KUKA KRL program: f1_Kuka_APT208T03S08.SRC

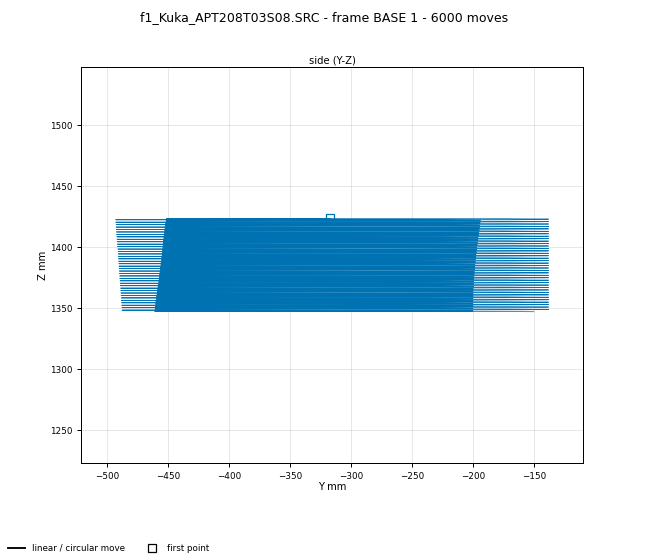
[picture p0: tool path of f1_Kuka_APT208T03S08.SRC in frame BASE 1, 6000 of 6001 moves have a stored position in this frame; points joined in program order, loops and branches not executed]
&ACCESS RVP
&REL 2
&PARAM TEMPLATE = C:\KRC\Roboter\Template\vorgabe
&PARAM EDITMASK = *
DEF f1_Kuka_APT208T03S08()


;FOLD INI;%{PE}%V3.2.0,%MKUKATPBASIS,%CINIT,%VCOMMON,%P
  ;FOLD BAS INI;%{E}%V3.2.0,%MKUKATPBASIS,%CINIT,%VINIT,%P
    GLOBAL INTERRUPT DECL 3 WHEN $STOPMESS==TRUE DO IR_STOPM ( )
    INTERRUPT ON 3
    BAS (#INITMOV,0 )
  ;ENDFOLD (BAS INI)
  ;FOLD USER INI;%{E}%V3.2.0,%MKUKATPUSER,%CINIT,%VINIT,%P
    ;Make your modifications here
  ;ENDFOLD (USER INI)
;ENDFOLD (INI)


;*** Make Null PTP Move
  PTP $pos_act

;*** Auto Load The Correct TOOL Data
  $tool=tool_data[3]

;*** Auto Load The Correct BASE Data
  $base=base_data[1]

  $ADVANCE = 5

;*** Restate Last Velocity
MMPM(30000.0)
SetRPM(6000)
LIN {X 0.078,Y -317.280,Z 1423.657,A 0.000,B 0.000,C 90.000,E1 298.281} C_DIS
LIN {X 0.027,Y -327.861,Z 1423.650,A 0.000,B 0.000,C 90.000,E1 297.052} C_DIS
LIN {X 0.042,Y -349.398,Z 1423.638,A 0.000,B 0.000,C 90.000,E1 294.771} C_DIS
LIN {X 0.137,Y -360.246,Z 1423.631,A 0.000,B 0.000,C 90.000,E1 293.643} C_DIS
LIN {X -0.205,Y -370.701,Z 1423.625,A 0.000,B 0.000,C 90.000,E1 292.589} C_DIS
LIN {X -0.139,Y -380.922,Z 1423.619,A 0.000,B 0.000,C 90.000,E1 291.461} C_DIS
LIN {X 0.117,Y -393.713,Z 1423.611,A 0.000,B 0.000,C 90.000,E1 289.993} C_DIS
LIN {X 0.075,Y -408.828,Z 1423.602,A 0.000,B 0.000,C 90.000,E1 288.308} C_DIS
LIN {X 0.018,Y -418.717,Z 1423.596,A 0.000,B 0.000,C 90.000,E1 287.221} C_DIS
LIN {X 0.155,Y -425.616,Z 1423.591,A 0.000,B 0.000,C 90.000,E1 286.386} C_DIS
LIN {X -0.080,Y -431.756,Z 1423.587,A 0.000,B 0.000,C 90.000,E1 285.607} C_DIS
LIN {X 0.159,Y -436.943,Z 1423.582,A 0.000,B 0.000,C 90.000,E1 284.773} C_DIS
LIN {X -0.092,Y -441.232,Z 1423.578,A 0.000,B 0.000,C 90.000,E1 284.008} C_DIS
LIN {X 0.232,Y -444.816,Z 1423.573,A 0.000,B 0.000,C 90.000,E1 283.175} C_DIS
LIN {X 0.051,Y -447.674,Z 1423.569,A 0.000,B 0.000,C 90.000,E1 282.411} C_DIS
LIN {X 0.083,Y -449.182,Z 1423.566,A 0.000,B 0.000,C 90.000,E1 281.883} C_DIS
LIN {X 0.037,Y -450.321,Z 1423.563,A 0.000,B 0.000,C 90.000,E1 281.366} C_DIS
LIN {X 0.091,Y -451.038,Z 1423.560,A 0.000,B 0.000,C 90.000,E1 280.838} C_DIS
LIN {X 0.150,Y -451.344,Z 1423.557,A 0.000,B 0.000,C 90.000,E1 280.310} C_DIS
LIN {X 0.133,Y -451.155,Z 1423.554,A 0.000,B 0.000,C 90.000,E1 279.792} C_DIS
LIN {X 0.195,Y -450.506,Z 1423.552,A 0.000,B 0.000,C 90.000,E1 279.265} C_DIS
LIN {X 0.182,Y -449.231,Z 1423.549,A 0.000,B 0.000,C 90.000,E1 278.746} C_DIS
LIN {X 0.234,Y -447.401,Z 1423.546,A 0.000,B 0.000,C 90.000,E1 278.219} C_DIS
LIN {X 0.210,Y -444.863,Z 1423.543,A 0.000,B 0.000,C 90.000,E1 277.701} C_DIS
LIN {X 0.172,Y -441.534,Z 1423.540,A 0.000,B 0.000,C 90.000,E1 277.182} C_DIS
LIN {X -0.047,Y -439.509,Z 1423.539,A 0.000,B 0.000,C 90.000,E1 276.947} C_DIS
LIN {X -0.110,Y -434.621,Z 1423.536,A 0.000,B 0.000,C 90.000,E1 276.429} C_DIS
LIN {X 0.045,Y -431.742,Z 1423.534,A 0.000,B 0.000,C 90.000,E1 276.144} C_DIS
LIN {X -0.110,Y -425.505,Z 1423.531,A 0.000,B 0.000,C 90.000,E1 275.682} C_DIS
LIN {X -0.196,Y -419.121,Z 1423.529,A 0.000,B 0.000,C 90.000,E1 275.277} C_DIS
LIN {X 0.069,Y -412.601,Z 1423.527,A 0.000,B 0.000,C 90.000,E1 274.878} C_DIS
LIN {X 0.054,Y -402.831,Z 1423.525,A 0.000,B 0.000,C 90.000,E1 274.416} C_DIS
LIN {X -0.018,Y -389.852,Z 1423.522,A 0.000,B 0.000,C 90.000,E1 273.898} C_DIS
LIN {X -0.100,Y -377.007,Z 1423.519,A 0.000,B 0.000,C 90.000,E1 273.440} C_DIS
LIN {X 0.045,Y -367.072,Z 1423.517,A 0.000,B 0.000,C 90.000,E1 273.094} C_DIS
LIN {X 0.073,Y -356.749,Z 1423.516,A 0.000,B 0.000,C 90.000,E1 272.808} C_DIS
LIN {X 0.056,Y -346.151,Z 1423.514,A 0.000,B 0.000,C 90.000,E1 272.579} C_DIS
LIN {X -0.061,Y -333.748,Z 1423.513,A 0.000,B 0.000,C 90.000,E1 272.407} C_DIS
LIN {X -0.117,Y -320.521,Z 1423.513,A 0.000,B 0.000,C 90.000,E1 272.293} C_DIS
LIN {X -0.070,Y -307.150,Z 1423.512,A 0.000,B 0.000,C 90.000,E1 272.236} C_DIS
LIN {X -0.069,Y -181.228,Z 1423.512,A 0.000,B 0.000,C 90.000,E1 272.236} C_DIS
LIN {X -0.066,Y -181.566,Z 1423.503,A 0.000,B 0.000,C 90.000,E1 270.516} C_DIS
LIN {X -0.076,Y -181.120,Z 1423.489,A 0.000,B 0.000,C 90.000,E1 267.993} C_DIS
LIN {X -0.088,Y -180.906,Z 1423.475,A 0.000,B 0.000,C 90.000,E1 265.469} C_DIS
LIN {X -0.031,Y -180.723,Z 1423.470,A 0.000,B 0.000,C 90.000,E1 264.609} C_DIS
LIN {X 0.066,Y -178.812,Z 1423.442,A 0.000,B 0.000,C 90.000,E1 259.511} C_DIS
LIN {X -0.026,Y -175.857,Z 1423.414,A 0.000,B 0.000,C 90.000,E1 254.448} C_DIS
LIN {X -0.045,Y -173.185,Z 1423.395,A 0.000,B 0.000,C 90.000,E1 251.040} C_DIS
LIN {X -0.042,Y -171.487,Z 1423.380,A 0.000,B 0.000,C 90.000,E1 248.465} C_DIS
LIN {X -0.054,Y -167.717,Z 1423.356,A 0.000,B 0.000,C 90.000,E1 244.152} C_DIS
LIN {X -0.038,Y -166.407,Z 1423.347,A 0.000,B 0.000,C 90.000,E1 242.410} C_DIS
LIN {X -0.040,Y -163.131,Z 1423.327,A 0.000,B 0.000,C 90.000,E1 238.918} C_DIS
LIN {X -0.074,Y -161.084,Z 1423.313,A 0.000,B 0.000,C 90.000,E1 236.294} C_DIS
LIN {X 0.036,Y -157.814,Z 1423.293,A 0.000,B 0.000,C 90.000,E1 232.718} C_DIS
LIN {X -0.026,Y -155.848,Z 1423.278,A 0.000,B 0.000,C 90.000,E1 230.070} C_DIS
LIN {X 0.031,Y -152.099,Z 1423.253,A 0.000,B 0.000,C 90.000,E1 225.567} C_DIS
LIN {X 0.049,Y -150.349,Z 1423.238,A 0.000,B 0.000,C 90.000,E1 222.852} C_DIS
LIN {X -0.022,Y -147.086,Z 1423.213,A 0.000,B 0.000,C 90.000,E1 218.338} C_DIS
LIN {X -0.027,Y -145.658,Z 1423.198,A 0.000,B 0.000,C 90.000,E1 215.598} C_DIS
LIN {X -0.024,Y -143.040,Z 1423.172,A 0.000,B 0.000,C 90.000,E1 211.003} C_DIS
LIN {X -0.023,Y -141.664,Z 1423.152,A 0.000,B 0.000,C 90.000,E1 207.308} C_DIS
LIN {X 0.022,Y -139.449,Z 1423.116,A 0.000,B 0.000,C 90.000,E1 200.791} C_DIS
LIN {X -0.058,Y -139.184,Z 1423.105,A 0.000,B 0.000,C 90.000,E1 198.960} C_DIS
LIN {X -0.034,Y -138.322,Z 1423.053,A 0.000,B 0.000,C 90.000,E1 189.613} C_DIS
LIN {X -0.027,Y -139.462,Z 1423.007,A 0.000,B 0.000,C 90.000,E1 181.203} C_DIS
LIN {X 0.053,Y -141.022,Z 1422.976,A 0.000,B 0.000,C 90.000,E1 175.584} C_DIS
LIN {X 0.007,Y -142.386,Z 1422.960,A 0.000,B 0.000,C 90.000,E1 172.818} C_DIS
LIN {X -0.072,Y -144.617,Z 1422.934,A 0.000,B 0.000,C 90.000,E1 168.229} C_DIS
LIN {X -0.010,Y -147.812,Z 1422.909,A 0.000,B 0.000,C 90.000,E1 163.614} C_DIS
LIN {X 0.077,Y -150.499,Z 1422.889,A 0.000,B 0.000,C 90.000,E1 159.934} C_DIS
LIN {X -0.043,Y -153.958,Z 1422.869,A 0.000,B 0.000,C 90.000,E1 156.357} C_DIS
LIN {X 0.019,Y -157.369,Z 1422.849,A 0.000,B 0.000,C 90.000,E1 152.743} C_DIS
LIN {X -0.038,Y -161.569,Z 1422.829,A 0.000,B 0.000,C 90.000,E1 149.203} C_DIS
LIN {X -0.027,Y -165.767,Z 1422.809,A 0.000,B 0.000,C 90.000,E1 145.674} C_DIS
LIN {X -0.040,Y -170.725,Z 1422.790,A 0.000,B 0.000,C 90.000,E1 142.190} C_DIS
LIN {X 0.002,Y -175.598,Z 1422.771,A 0.000,B 0.000,C 90.000,E1 138.728} C_DIS
LIN {X -0.011,Y -181.215,Z 1422.752,A 0.000,B 0.000,C 90.000,E1 135.324} C_DIS
LIN {X -0.019,Y -186.679,Z 1422.733,A 0.000,B 0.000,C 90.000,E1 131.962} C_DIS
LIN {X -0.075,Y -191.282,Z 1422.719,A 0.000,B 0.000,C 90.000,E1 129.483} C_DIS
LIN {X 0.005,Y -197.107,Z 1422.701,A 0.000,B 0.000,C 90.000,E1 126.171} C_DIS
LIN {X 0.026,Y -199.962,Z 1422.693,A 0.000,B 0.000,C 90.000,E1 124.739} C_DIS
LIN {X 0.006,Y -311.159,Z 1422.693,A 0.000,B 0.000,C 90.000,E1 124.739} C_DIS
LIN {X -0.064,Y -312.139,Z 1422.693,A 0.000,B 0.000,C 90.000,E1 124.739} C_DIS
LIN {X 0.065,Y -316.789,Z 1422.692,A 0.000,B 0.000,C 90.000,E1 124.532} C_DIS
LIN {X 0.109,Y -319.895,Z 1422.691,A 0.000,B 0.000,C 90.000,E1 124.278} C_DIS
LIN {X 0.005,Y -323.594,Z 1422.688,A 0.000,B 0.000,C 90.000,E1 123.833} C_DIS
LIN {X 0.086,Y -325.369,Z 1422.686,A 0.000,B 0.000,C 90.000,E1 123.499} C_DIS
LIN {X 0.169,Y -326.751,Z 1422.684,A 0.000,B 0.000,C 90.000,E1 123.166} C_DIS
LIN {X 0.039,Y -338.501,Z 1422.667,A 0.000,B 0.000,C 90.000,E1 120.050} C_DIS
LIN {X 0.192,Y -350.479,Z 1422.652,A 0.000,B 0.000,C 90.000,E1 117.257} C_DIS
LIN {X -0.102,Y -363.919,Z 1422.636,A 0.000,B 0.000,C 90.000,E1 114.591} C_DIS
LIN {X 0.056,Y -377.182,Z 1422.623,A 0.000,B 0.000,C 90.000,E1 112.206} C_DIS
LIN {X 0.128,Y -391.780,Z 1422.611,A 0.000,B 0.000,C 90.000,E1 109.885} C_DIS
LIN {X 0.065,Y -407.816,Z 1422.598,A 0.000,B 0.000,C 90.000,E1 107.638} C_DIS
LIN {X 0.145,Y -425.401,Z 1422.586,A 0.000,B 0.000,C 90.000,E1 105.426} C_DIS
LIN {X 0.053,Y -444.616,Z 1422.574,A 0.000,B 0.000,C 90.000,E1 103.300} C_DIS
LIN {X 0.107,Y -464.726,Z 1422.563,A 0.000,B 0.000,C 90.000,E1 101.299} C_DIS
LIN {X -0.177,Y -485.356,Z 1422.553,A 0.000,B 0.000,C 90.000,E1 99.500} C_DIS
LIN {X -0.056,Y -487.492,Z 1422.551,A 0.000,B 0.000,C 90.000,E1 99.265} C_DIS
LIN {X 0.065,Y -489.116,Z 1422.550,A 0.000,B 0.000,C 90.000,E1 99.029} C_DIS
LIN {X -0.113,Y -490.499,Z 1422.549,A 0.000,B 0.000,C 90.000,E1 98.803} C_DIS
LIN {X -0.215,Y -491.522,Z 1422.547,A 0.000,B 0.000,C 90.000,E1 98.568} C_DIS
LIN {X 0.009,Y -492.685,Z 1422.545,A 0.000,B 0.000,C 90.000,E1 98.049} C_DIS
LIN {X -0.247,Y -492.827,Z 1422.542,A 0.000,B 0.000,C 90.000,E1 97.587} C_DIS
LIN {X -0.007,Y -491.972,Z 1422.539,A 0.000,B 0.000,C 90.000,E1 97.068} C_DIS
LIN {X -0.253,Y -489.975,Z 1422.536,A 0.000,B 0.000,C 90.000,E1 96.606} C_DIS
LIN {X 0.196,Y -483.357,Z 1422.531,A 0.000,B 0.000,C 90.000,E1 95.568} C_DIS
LIN {X 0.126,Y -469.087,Z 1422.519,A 0.000,B 0.000,C 90.000,E1 93.326} C_DIS
LIN {X 0.072,Y -460.783,Z 1422.511,A 0.000,B 0.000,C 90.000,E1 92.064} C_DIS
LIN {X -0.021,Y -440.905,Z 1422.494,A 0.000,B 0.000,C 90.000,E1 88.969} C_DIS
LIN {X -0.162,Y -429.949,Z 1422.484,A 0.000,B 0.000,C 90.000,E1 87.135} C_DIS
LIN {X -0.076,Y -418.773,Z 1422.474,A 0.000,B 0.000,C 90.000,E1 85.241} C_DIS
LIN {X -0.085,Y -405.939,Z 1422.461,A 0.000,B 0.000,C 90.000,E1 83.053} C_DIS
LIN {X 0.034,Y -394.598,Z 1422.450,A 0.000,B 0.000,C 90.000,E1 81.084} C_DIS
LIN {X -0.016,Y -383.087,Z 1422.439,A 0.000,B 0.000,C 90.000,E1 79.106} C_DIS
LIN {X 0.130,Y -371.680,Z 1422.428,A 0.000,B 0.000,C 90.000,E1 77.061} C_DIS
LIN {X -0.149,Y -360.358,Z 1422.417,A 0.000,B 0.000,C 90.000,E1 75.046} C_DIS
LIN {X 0.121,Y -349.003,Z 1422.405,A 0.000,B 0.000,C 90.000,E1 72.906} C_DIS
LIN {X 0.016,Y -339.072,Z 1422.395,A 0.000,B 0.000,C 90.000,E1 71.094} C_DIS
LIN {X 0.102,Y -325.927,Z 1422.381,A 0.000,B 0.000,C 90.000,E1 68.592} C_DIS
LIN {X -0.007,Y -308.641,Z 1422.362,A 0.000,B 0.000,C 90.000,E1 65.101} C_DIS
LIN {X -0.028,Y -295.960,Z 1422.345,A 0.000,B 0.000,C 90.000,E1 62.153} C_DIS
LIN {X 0.004,Y -283.341,Z 1422.327,A 0.000,B 0.000,C 90.000,E1 58.791} C_DIS
LIN {X -0.145,Y -271.830,Z 1422.307,A 0.000,B 0.000,C 90.000,E1 55.388} C_DIS
LIN {X 0.077,Y -262.146,Z 1422.290,A 0.000,B 0.000,C 90.000,E1 52.190} C_DIS
LIN {X -0.025,Y -252.090,Z 1422.270,A 0.000,B 0.000,C 90.000,E1 48.647} C_DIS
LIN {X 0.025,Y -242.796,Z 1422.250,A 0.000,B 0.000,C 90.000,E1 45.000} C_DIS
LIN {X -0.027,Y -234.404,Z 1422.229,A 0.000,B 0.000,C 90.000,E1 41.310} C_DIS
LIN {X 0.060,Y -226.842,Z 1422.208,A 0.000,B 0.000,C 90.000,E1 37.523} C_DIS
LIN {X 0.036,Y -220.187,Z 1422.187,A 0.000,B 0.000,C 90.000,E1 33.706} C_DIS
LIN {X -0.122,Y -214.311,Z 1422.166,A 0.000,B 0.000,C 90.000,E1 29.873} C_DIS
LIN {X -0.025,Y -209.279,Z 1422.144,A 0.000,B 0.000,C 90.000,E1 25.924} C_DIS
LIN {X -0.066,Y -205.139,Z 1422.122,A 0.000,B 0.000,C 90.000,E1 21.972} C_DIS
LIN {X 0.010,Y -201.303,Z 1422.095,A 0.000,B 0.000,C 90.000,E1 17.149} C_DIS
LIN {X 0.047,Y -198.459,Z 1422.068,A 0.000,B 0.000,C 90.000,E1 12.299} C_DIS
LIN {X 0.088,Y -196.155,Z 1422.037,A 0.000,B 0.000,C 90.000,E1 6.606} C_DIS
LIN {X 0.027,Y -194.653,Z 1422.005,A 0.000,B 0.000,C 90.000,E1 0.917} C_DIS
LIN {X 0.004,Y -194.202,Z 1421.984,A 0.000,B 0.000,C 90.000,E1 357.078} C_DIS
LIN {X -0.051,Y -194.204,Z 1421.957,A 0.000,B 0.000,C 90.000,E1 352.186} C_DIS
LIN {X -0.046,Y -195.369,Z 1421.920,A 0.000,B 0.000,C 90.000,E1 345.644} C_DIS
LIN {X -0.018,Y -198.094,Z 1421.889,A 0.000,B 0.000,C 90.000,E1 339.934} C_DIS
LIN {X -0.100,Y -202.039,Z 1421.862,A 0.000,B 0.000,C 90.000,E1 335.101} C_DIS
LIN {X 0.034,Y -206.546,Z 1421.839,A 0.000,B 0.000,C 90.000,E1 331.051} C_DIS
LIN {X 0.048,Y -210.949,Z 1421.822,A 0.000,B 0.000,C 90.000,E1 327.867} C_DIS
LIN {X -0.018,Y -216.341,Z 1421.804,A 0.000,B 0.000,C 90.000,E1 324.736} C_DIS
LIN {X 0.002,Y -222.667,Z 1421.787,A 0.000,B 0.000,C 90.000,E1 321.618} C_DIS
LIN {X -0.075,Y -229.928,Z 1421.770,A 0.000,B 0.000,C 90.000,E1 318.566} C_DIS
LIN {X -0.029,Y -239.211,Z 1421.751,A 0.000,B 0.000,C 90.000,E1 315.162} C_DIS
LIN {X -0.040,Y -249.686,Z 1421.732,A 0.000,B 0.000,C 90.000,E1 311.838} C_DIS
LIN {X 0.098,Y -260.059,Z 1421.716,A 0.000,B 0.000,C 90.000,E1 308.910} C_DIS
LIN {X 0.021,Y -271.627,Z 1421.701,A 0.000,B 0.000,C 90.000,E1 306.091} C_DIS
LIN {X 0.083,Y -281.387,Z 1421.689,A 0.000,B 0.000,C 90.000,E1 303.992} C_DIS
LIN {X 0.073,Y -288.584,Z 1421.681,A 0.000,B 0.000,C 90.000,E1 302.625} C_DIS
LIN {X 0.154,Y -296.526,Z 1421.674,A 0.000,B 0.000,C 90.000,E1 301.258} C_DIS
LIN {X 0.029,Y -305.181,Z 1421.666,A 0.000,B 0.000,C 90.000,E1 299.951} C_DIS
LIN {X 0.166,Y -314.744,Z 1421.659,A 0.000,B 0.000,C 90.000,E1 298.615} C_DIS
LIN {X 0.045,Y -325.085,Z 1421.652,A 0.000,B 0.000,C 90.000,E1 297.385} C_DIS
LIN {X 0.084,Y -346.523,Z 1421.639,A 0.000,B 0.000,C 90.000,E1 295.079} C_DIS
LIN {X 0.154,Y -359.883,Z 1421.632,A 0.000,B 0.000,C 90.000,E1 293.695} C_DIS
LIN {X -0.165,Y -370.313,Z 1421.626,A 0.000,B 0.000,C 90.000,E1 292.642} C_DIS
LIN {X 0.087,Y -380.561,Z 1421.619,A 0.000,B 0.000,C 90.000,E1 291.482} C_DIS
LIN {X 0.001,Y -393.292,Z 1421.611,A 0.000,B 0.000,C 90.000,E1 290.066} C_DIS
LIN {X 0.132,Y -408.362,Z 1421.602,A 0.000,B 0.000,C 90.000,E1 288.362} C_DIS
LIN {X -0.004,Y -418.330,Z 1421.596,A 0.000,B 0.000,C 90.000,E1 287.275} C_DIS
LIN {X -0.191,Y -425.234,Z 1421.592,A 0.000,B 0.000,C 90.000,E1 286.496} C_DIS
LIN {X -0.022,Y -431.464,Z 1421.587,A 0.000,B 0.000,C 90.000,E1 285.662} C_DIS
LIN {X -0.089,Y -435.100,Z 1421.584,A 0.000,B 0.000,C 90.000,E1 285.134} C_DIS
LIN {X 0.182,Y -439.765,Z 1421.580,A 0.000,B 0.000,C 90.000,E1 284.300} C_DIS
LIN {X -0.044,Y -443.624,Z 1421.575,A 0.000,B 0.000,C 90.000,E1 283.536} C_DIS
LIN {X -0.029,Y -445.806,Z 1421.572,A 0.000,B 0.000,C 90.000,E1 283.008} C_DIS
LIN {X 0.001,Y -447.703,Z 1421.569,A 0.000,B 0.000,C 90.000,E1 282.479} C_DIS
LIN {X 0.037,Y -449.267,Z 1421.566,A 0.000,B 0.000,C 90.000,E1 281.951} C_DIS
LIN {X 0.082,Y -450.452,Z 1421.563,A 0.000,B 0.000,C 90.000,E1 281.422} C_DIS
LIN {X 0.137,Y -451.260,Z 1421.561,A 0.000,B 0.000,C 90.000,E1 280.894} C_DIS
LIN {X 0.196,Y -451.636,Z 1421.558,A 0.000,B 0.000,C 90.000,E1 280.366} C_DIS
LIN {X 0.179,Y -451.549,Z 1421.555,A 0.000,B 0.000,C 90.000,E1 279.849} C_DIS
LIN {X 0.242,Y -450.932,Z 1421.552,A 0.000,B 0.000,C 90.000,E1 279.321} C_DIS
LIN {X -0.214,Y -449.794,Z 1421.549,A 0.000,B 0.000,C 90.000,E1 278.859} C_DIS
LIN {X -0.224,Y -448.053,Z 1421.546,A 0.000,B 0.000,C 90.000,E1 278.341} C_DIS
LIN {X -0.178,Y -445.618,Z 1421.543,A 0.000,B 0.000,C 90.000,E1 277.814} C_DIS
LIN {X -0.210,Y -442.391,Z 1421.540,A 0.000,B 0.000,C 90.000,E1 277.296} C_DIS
LIN {X 0.011,Y -440.500,Z 1421.539,A 0.000,B 0.000,C 90.000,E1 277.004} C_DIS
LIN {X -0.049,Y -435.790,Z 1421.536,A 0.000,B 0.000,C 90.000,E1 276.486} C_DIS
LIN {X 0.109,Y -433.033,Z 1421.535,A 0.000,B 0.000,C 90.000,E1 276.201} C_DIS
LIN {X -0.144,Y -426.825,Z 1421.532,A 0.000,B 0.000,C 90.000,E1 275.739} C_DIS
LIN {X 0.107,Y -420.413,Z 1421.529,A 0.000,B 0.000,C 90.000,E1 275.277} C_DIS
LIN {X -0.107,Y -413.942,Z 1421.527,A 0.000,B 0.000,C 90.000,E1 274.935} C_DIS
LIN {X 0.054,Y -407.470,Z 1421.526,A 0.000,B 0.000,C 90.000,E1 274.588} C_DIS
LIN {X -0.116,Y -397.720,Z 1421.523,A 0.000,B 0.000,C 90.000,E1 274.188} C_DIS
LIN {X 0.001,Y -384.828,Z 1421.520,A 0.000,B 0.000,C 90.000,E1 273.669} C_DIS
LIN {X 0.050,Y -371.840,Z 1421.518,A 0.000,B 0.000,C 90.000,E1 273.212} C_DIS
LIN {X -0.033,Y -361.640,Z 1421.516,A 0.000,B 0.000,C 90.000,E1 272.922} C_DIS
LIN {X -0.159,Y -350.920,Z 1421.515,A 0.000,B 0.000,C 90.000,E1 272.694} C_DIS
LIN {X 0.014,Y -343.452,Z 1421.514,A 0.000,B 0.000,C 90.000,E1 272.522} C_DIS
LIN {X -0.054,Y -335.045,Z 1421.513,A 0.000,B 0.000,C 90.000,E1 272.407} C_DIS
LIN {X -0.110,Y -321.941,Z 1421.513,A 0.000,B 0.000,C 90.000,E1 272.293} C_DIS
LIN {X -0.069,Y -310.020,Z 1421.512,A 0.000,B 0.000,C 90.000,E1 272.236} C_DIS
LIN {X -0.069,Y -181.228,Z 1421.512,A 0.000,B 0.000,C 90.000,E1 272.236} C_DIS
LIN {X -0.072,Y -181.566,Z 1421.503,A 0.000,B 0.000,C 90.000,E1 270.516} C_DIS
LIN {X -0.082,Y -181.119,Z 1421.489,A 0.000,B 0.000,C 90.000,E1 267.993} C_DIS
LIN {X 0.087,Y -180.907,Z 1421.475,A 0.000,B 0.000,C 90.000,E1 265.412} C_DIS
LIN {X -0.036,Y -180.723,Z 1421.470,A 0.000,B 0.000,C 90.000,E1 264.609} C_DIS
LIN {X 0.061,Y -178.811,Z 1421.442,A 0.000,B 0.000,C 90.000,E1 259.511} C_DIS
LIN {X -0.032,Y -175.856,Z 1421.414,A 0.000,B 0.000,C 90.000,E1 254.448} C_DIS
LIN {X -0.050,Y -173.184,Z 1421.395,A 0.000,B 0.000,C 90.000,E1 251.040} C_DIS
LIN {X -0.048,Y -171.486,Z 1421.380,A 0.000,B 0.000,C 90.000,E1 248.465} C_DIS
LIN {X -0.060,Y -167.715,Z 1421.356,A 0.000,B 0.000,C 90.000,E1 244.152} C_DIS
LIN {X -0.044,Y -166.406,Z 1421.347,A 0.000,B 0.000,C 90.000,E1 242.410} C_DIS
LIN {X -0.045,Y -163.130,Z 1421.327,A 0.000,B 0.000,C 90.000,E1 238.918} C_DIS
LIN {X -0.079,Y -161.082,Z 1421.313,A 0.000,B 0.000,C 90.000,E1 236.294} C_DIS
LIN {X 0.031,Y -157.812,Z 1421.293,A 0.000,B 0.000,C 90.000,E1 232.718} C_DIS
LIN {X -0.031,Y -155.847,Z 1421.278,A 0.000,B 0.000,C 90.000,E1 230.070} C_DIS
LIN {X 0.025,Y -152.097,Z 1421.253,A 0.000,B 0.000,C 90.000,E1 225.567} C_DIS
LIN {X 0.044,Y -150.348,Z 1421.238,A 0.000,B 0.000,C 90.000,E1 222.852} C_DIS
LIN {X -0.027,Y -147.085,Z 1421.213,A 0.000,B 0.000,C 90.000,E1 218.338} C_DIS
LIN {X -0.032,Y -145.657,Z 1421.198,A 0.000,B 0.000,C 90.000,E1 215.598} C_DIS
LIN {X -0.029,Y -143.040,Z 1421.172,A 0.000,B 0.000,C 90.000,E1 211.003} C_DIS
LIN {X -0.028,Y -141.664,Z 1421.152,A 0.000,B 0.000,C 90.000,E1 207.308} C_DIS
LIN {X 0.017,Y -139.449,Z 1421.116,A 0.000,B 0.000,C 90.000,E1 200.791} C_DIS
LIN {X 0.069,Y -139.183,Z 1421.105,A 0.000,B 0.000,C 90.000,E1 198.906} C_DIS
LIN {X -0.039,Y -138.321,Z 1421.053,A 0.000,B 0.000,C 90.000,E1 189.613} C_DIS
LIN {X -0.032,Y -139.463,Z 1421.007,A 0.000,B 0.000,C 90.000,E1 181.203} C_DIS
LIN {X 0.048,Y -141.023,Z 1420.976,A 0.000,B 0.000,C 90.000,E1 175.584} C_DIS
LIN {X 0.003,Y -142.387,Z 1420.960,A 0.000,B 0.000,C 90.000,E1 172.818} C_DIS
LIN {X 0.065,Y -144.619,Z 1420.934,A 0.000,B 0.000,C 90.000,E1 168.173} C_DIS
LIN {X -0.015,Y -147.812,Z 1420.909,A 0.000,B 0.000,C 90.000,E1 163.614} C_DIS
LIN {X 0.073,Y -150.501,Z 1420.889,A 0.000,B 0.000,C 90.000,E1 159.934} C_DIS
LIN {X -0.048,Y -153.960,Z 1420.869,A 0.000,B 0.000,C 90.000,E1 156.357} C_DIS
LIN {X 0.015,Y -157.371,Z 1420.849,A 0.000,B 0.000,C 90.000,E1 152.743} C_DIS
LIN {X -0.044,Y -161.572,Z 1420.829,A 0.000,B 0.000,C 90.000,E1 149.203} C_DIS
LIN {X -0.032,Y -165.769,Z 1420.809,A 0.000,B 0.000,C 90.000,E1 145.674} C_DIS
LIN {X -0.045,Y -170.728,Z 1420.790,A 0.000,B 0.000,C 90.000,E1 142.190} C_DIS
LIN {X -0.002,Y -175.600,Z 1420.771,A 0.000,B 0.000,C 90.000,E1 138.728} C_DIS
LIN {X -0.016,Y -181.217,Z 1420.752,A 0.000,B 0.000,C 90.000,E1 135.324} C_DIS
LIN {X -0.024,Y -186.683,Z 1420.733,A 0.000,B 0.000,C 90.000,E1 131.962} C_DIS
LIN {X -0.081,Y -191.285,Z 1420.719,A 0.000,B 0.000,C 90.000,E1 129.483} C_DIS
LIN {X -0.001,Y -197.110,Z 1420.701,A 0.000,B 0.000,C 90.000,E1 126.171} C_DIS
LIN {X -0.021,Y -199.922,Z 1420.693,A 0.000,B 0.000,C 90.000,E1 124.771} C_DIS
LIN {X 0.108,Y -311.246,Z 1420.693,A 0.000,B 0.000,C 90.000,E1 124.739} C_DIS
LIN {X 0.056,Y -317.044,Z 1420.692,A 0.000,B 0.000,C 90.000,E1 124.532} C_DIS
LIN {X 0.084,Y -320.054,Z 1420.691,A 0.000,B 0.000,C 90.000,E1 124.278} C_DIS
LIN {X 0.154,Y -323.760,Z 1420.688,A 0.000,B 0.000,C 90.000,E1 123.785} C_DIS
LIN {X -0.033,Y -325.477,Z 1420.686,A 0.000,B 0.000,C 90.000,E1 123.499} C_DIS
LIN {X -0.125,Y -327.926,Z 1420.682,A 0.000,B 0.000,C 90.000,E1 122.880} C_DIS
LIN {X -0.082,Y -338.563,Z 1420.667,A 0.000,B 0.000,C 90.000,E1 120.050} C_DIS
LIN {X 0.067,Y -350.550,Z 1420.651,A 0.000,B 0.000,C 90.000,E1 117.257} C_DIS
LIN {X -0.077,Y -364.001,Z 1420.636,A 0.000,B 0.000,C 90.000,E1 114.567} C_DIS
LIN {X -0.073,Y -377.275,Z 1420.623,A 0.000,B 0.000,C 90.000,E1 112.206} C_DIS
LIN {X -0.003,Y -391.885,Z 1420.610,A 0.000,B 0.000,C 90.000,E1 109.885} C_DIS
LIN {X -0.070,Y -407.932,Z 1420.598,A 0.000,B 0.000,C 90.000,E1 107.638} C_DIS
LIN {X 0.007,Y -425.531,Z 1420.586,A 0.000,B 0.000,C 90.000,E1 105.426} C_DIS
LIN {X -0.086,Y -444.758,Z 1420.574,A 0.000,B 0.000,C 90.000,E1 103.300} C_DIS
LIN {X -0.027,Y -464.873,Z 1420.563,A 0.000,B 0.000,C 90.000,E1 101.299} C_DIS
LIN {X 0.172,Y -485.485,Z 1420.553,A 0.000,B 0.000,C 90.000,E1 99.443} C_DIS
LIN {X -0.196,Y -487.560,Z 1420.551,A 0.000,B 0.000,C 90.000,E1 99.265} C_DIS
LIN {X -0.085,Y -489.142,Z 1420.550,A 0.000,B 0.000,C 90.000,E1 99.029} C_DIS
LIN {X -0.263,Y -490.481,Z 1420.549,A 0.000,B 0.000,C 90.000,E1 98.803} C_DIS
LIN {X 0.120,Y -491.469,Z 1420.547,A 0.000,B 0.000,C 90.000,E1 98.511} C_DIS
LIN {X -0.142,Y -492.573,Z 1420.545,A 0.000,B 0.000,C 90.000,E1 98.049} C_DIS
LIN {X 0.091,Y -492.661,Z 1420.542,A 0.000,B 0.000,C 90.000,E1 97.530} C_DIS
LIN {X -0.158,Y -491.750,Z 1420.539,A 0.000,B 0.000,C 90.000,E1 97.068} C_DIS
LIN {X 0.082,Y -489.682,Z 1420.536,A 0.000,B 0.000,C 90.000,E1 96.549} C_DIS
LIN {X -0.119,Y -471.909,Z 1420.521,A 0.000,B 0.000,C 90.000,E1 93.841} C_DIS
LIN {X 0.066,Y -465.501,Z 1420.516,A 0.000,B 0.000,C 90.000,E1 92.808} C_DIS
LIN {X -0.035,Y -453.683,Z 1420.506,A 0.000,B 0.000,C 90.000,E1 91.031} C_DIS
LIN {X -0.087,Y -435.958,Z 1420.490,A 0.000,B 0.000,C 90.000,E1 88.165} C_DIS
LIN {X -0.159,Y -428.109,Z 1420.482,A 0.000,B 0.000,C 90.000,E1 86.846} C_DIS
LIN {X 0.177,Y -418.551,Z 1420.473,A 0.000,B 0.000,C 90.000,E1 85.184} C_DIS
LIN {X 0.153,Y -405.740,Z 1420.461,A 0.000,B 0.000,C 90.000,E1 82.996} C_DIS
LIN {X -0.203,Y -396.035,Z 1420.452,A 0.000,B 0.000,C 90.000,E1 81.376} C_DIS
LIN {X 0.112,Y -386.226,Z 1420.443,A 0.000,B 0.000,C 90.000,E1 79.634} C_DIS
LIN {X -0.034,Y -373.150,Z 1420.430,A 0.000,B 0.000,C 90.000,E1 77.353} C_DIS
LIN {X 0.069,Y -361.829,Z 1420.418,A 0.000,B 0.000,C 90.000,E1 75.283} C_DIS
LIN {X 0.036,Y -350.461,Z 1420.407,A 0.000,B 0.000,C 90.000,E1 73.196} C_DIS
LIN {X -0.144,Y -340.573,Z 1420.396,A 0.000,B 0.000,C 90.000,E1 71.402} C_DIS
LIN {X -0.018,Y -327.372,Z 1420.383,A 0.000,B 0.000,C 90.000,E1 68.901} C_DIS
LIN {X -0.077,Y -309.930,Z 1420.363,A 0.000,B 0.000,C 90.000,E1 65.409} C_DIS
LIN {X 0.075,Y -297.134,Z 1420.347,A 0.000,B 0.000,C 90.000,E1 62.436} C_DIS
LIN {X -0.098,Y -285.611,Z 1420.330,A 0.000,B 0.000,C 90.000,E1 59.459} C_DIS
LIN {X 0.056,Y -273.952,Z 1420.311,A 0.000,B 0.000,C 90.000,E1 56.008} C_DIS
LIN {X -0.034,Y -264.211,Z 1420.294,A 0.000,B 0.000,C 90.000,E1 52.889} C_DIS
LIN {X 0.137,Y -254.008,Z 1420.274,A 0.000,B 0.000,C 90.000,E1 49.299} C_DIS
LIN {X -0.090,Y -244.588,Z 1420.254,A 0.000,B 0.000,C 90.000,E1 45.729} C_DIS
LIN {X 0.077,Y -236.040,Z 1420.233,A 0.000,B 0.000,C 90.000,E1 42.000} C_DIS
LIN {X 0.036,Y -228.338,Z 1420.213,A 0.000,B 0.000,C 90.000,E1 38.257} C_DIS
LIN {X 0.009,Y -221.529,Z 1420.191,A 0.000,B 0.000,C 90.000,E1 34.452} C_DIS
LIN {X -0.002,Y -215.542,Z 1420.170,A 0.000,B 0.000,C 90.000,E1 30.590} C_DIS
LIN {X 0.036,Y -210.353,Z 1420.148,A 0.000,B 0.000,C 90.000,E1 26.668} C_DIS
LIN {X 0.019,Y -206.069,Z 1420.126,A 0.000,B 0.000,C 90.000,E1 22.717} C_DIS
LIN {X -0.055,Y -202.099,Z 1420.100,A 0.000,B 0.000,C 90.000,E1 17.946} C_DIS
LIN {X -0.070,Y -199.183,Z 1420.073,A 0.000,B 0.000,C 90.000,E1 13.119} C_DIS
LIN {X 0.069,Y -197.011,Z 1420.046,A 0.000,B 0.000,C 90.000,E1 8.219} C_DIS
LIN {X -0.018,Y -195.935,Z 1420.028,A 0.000,B 0.000,C 90.000,E1 4.992} C_DIS
LIN {X -0.035,Y -194.777,Z 1419.997,A 0.000,B 0.000,C 90.000,E1 359.542} C_DIS
LIN {X 0.067,Y -194.386,Z 1419.970,A 0.000,B 0.000,C 90.000,E1 354.609} C_DIS
LIN {X -0.054,Y -194.593,Z 1419.947,A 0.000,B 0.000,C 90.000,E1 350.557} C_DIS
LIN {X -0.011,Y -196.562,Z 1419.907,A 0.000,B 0.000,C 90.000,E1 343.196} C_DIS
LIN {X 0.079,Y -200.084,Z 1419.875,A 0.000,B 0.000,C 90.000,E1 337.486} C_DIS
LIN {X 0.064,Y -203.944,Z 1419.853,A 0.000,B 0.000,C 90.000,E1 333.461} C_DIS
LIN {X 0.091,Y -208.830,Z 1419.830,A 0.000,B 0.000,C 90.000,E1 329.459} C_DIS
LIN {X 0.096,Y -213.732,Z 1419.813,A 0.000,B 0.000,C 90.000,E1 326.294} C_DIS
LIN {X -0.081,Y -219.597,Z 1419.796,A 0.000,B 0.000,C 90.000,E1 323.210} C_DIS
LIN {X -0.061,Y -226.355,Z 1419.778,A 0.000,B 0.000,C 90.000,E1 320.114} C_DIS
LIN {X 0.054,Y -235.131,Z 1419.759,A 0.000,B 0.000,C 90.000,E1 316.662} C_DIS
LIN {X -0.058,Y -243.885,Z 1419.743,A 0.000,B 0.000,C 90.000,E1 313.704} C_DIS
LIN {X 0.082,Y -254.850,Z 1419.724,A 0.000,B 0.000,C 90.000,E1 310.378} C_DIS
LIN {X 0.089,Y -267.243,Z 1419.707,A 0.000,B 0.000,C 90.000,E1 307.156} C_DIS
LIN {X -0.159,Y -276.484,Z 1419.695,A 0.000,B 0.000,C 90.000,E1 305.105} C_DIS
LIN {X -0.129,Y -284.944,Z 1419.685,A 0.000,B 0.000,C 90.000,E1 303.372} C_DIS
LIN {X -0.113,Y -294.511,Z 1419.676,A 0.000,B 0.000,C 90.000,E1 301.671} C_DIS
LIN {X -0.105,Y -305.234,Z 1419.667,A 0.000,B 0.000,C 90.000,E1 300.001} C_DIS
LIN {X -0.126,Y -314.773,Z 1419.659,A 0.000,B 0.000,C 90.000,E1 298.693} C_DIS
LIN {X -0.023,Y -324.959,Z 1419.652,A 0.000,B 0.000,C 90.000,E1 297.436} C_DIS
LIN {X -0.114,Y -346.306,Z 1419.640,A 0.000,B 0.000,C 90.000,E1 295.155} C_DIS
LIN {X -0.145,Y -359.788,Z 1419.632,A 0.000,B 0.000,C 90.000,E1 293.770} C_DIS
LIN {X 0.005,Y -370.222,Z 1419.626,A 0.000,B 0.000,C 90.000,E1 292.642} C_DIS
LIN {X 0.180,Y -377.995,Z 1419.621,A 0.000,B 0.000,C 90.000,E1 291.770} C_DIS
LIN {X -0.053,Y -390.719,Z 1419.613,A 0.000,B 0.000,C 90.000,E1 290.375} C_DIS
LIN {X 0.076,Y -405.734,Z 1419.604,A 0.000,B 0.000,C 90.000,E1 288.671} C_DIS
LIN {X -0.043,Y -415.761,Z 1419.598,A 0.000,B 0.000,C 90.000,E1 287.583} C_DIS
LIN {X 0.163,Y -422.945,Z 1419.593,A 0.000,B 0.000,C 90.000,E1 286.732} C_DIS
LIN {X -0.092,Y -429.472,Z 1419.589,A 0.000,B 0.000,C 90.000,E1 285.953} C_DIS
LIN {X 0.002,Y -435.171,Z 1419.584,A 0.000,B 0.000,C 90.000,E1 285.134} C_DIS
LIN {X -0.151,Y -439.869,Z 1419.580,A 0.000,B 0.000,C 90.000,E1 284.356} C_DIS
LIN {X 0.051,Y -443.788,Z 1419.575,A 0.000,B 0.000,C 90.000,E1 283.536} C_DIS
LIN {X 0.067,Y -445.991,Z 1419.572,A 0.000,B 0.000,C 90.000,E1 283.008} C_DIS
LIN {X 0.098,Y -447.916,Z 1419.569,A 0.000,B 0.000,C 90.000,E1 282.479} C_DIS
LIN {X 0.135,Y -449.487,Z 1419.567,A 0.000,B 0.000,C 90.000,E1 281.951} C_DIS
LIN {X 0.183,Y -450.707,Z 1419.564,A 0.000,B 0.000,C 90.000,E1 281.422} C_DIS
LIN {X -0.205,Y -451.521,Z 1419.561,A 0.000,B 0.000,C 90.000,E1 280.950} C_DIS
LIN {X -0.145,Y -451.922,Z 1419.558,A 0.000,B 0.000,C 90.000,E1 280.423} C_DIS
LIN {X -0.161,Y -451.873,Z 1419.555,A 0.000,B 0.000,C 90.000,E1 279.905} C_DIS
LIN {X -0.096,Y -451.275,Z 1419.552,A 0.000,B 0.000,C 90.000,E1 279.378} C_DIS
LIN {X -0.105,Y -450.177,Z 1419.549,A 0.000,B 0.000,C 90.000,E1 278.859} C_DIS
LIN {X -0.115,Y -448.503,Z 1419.546,A 0.000,B 0.000,C 90.000,E1 278.341} C_DIS
LIN {X -0.067,Y -446.073,Z 1419.543,A 0.000,B 0.000,C 90.000,E1 277.814} C_DIS
LIN {X 0.108,Y -444.638,Z 1419.542,A 0.000,B 0.000,C 90.000,E1 277.530} C_DIS
LIN {X 0.125,Y -441.063,Z 1419.539,A 0.000,B 0.000,C 90.000,E1 277.004} C_DIS
LIN {X 0.067,Y -436.393,Z 1419.536,A 0.000,B 0.000,C 90.000,E1 276.486} C_DIS
LIN {X -0.206,Y -433.714,Z 1419.535,A 0.000,B 0.000,C 90.000,E1 276.258} C_DIS
LIN {X -0.096,Y -427.480,Z 1419.532,A 0.000,B 0.000,C 90.000,E1 275.739} C_DIS
LIN {X 0.150,Y -421.147,Z 1419.529,A 0.000,B 0.000,C 90.000,E1 275.277} C_DIS
LIN {X -0.098,Y -414.709,Z 1419.527,A 0.000,B 0.000,C 90.000,E1 274.935} C_DIS
LIN {X -0.006,Y -408.117,Z 1419.526,A 0.000,B 0.000,C 90.000,E1 274.588} C_DIS
LIN {X -0.179,Y -398.393,Z 1419.523,A 0.000,B 0.000,C 90.000,E1 274.188} C_DIS
LIN {X -0.066,Y -385.556,Z 1419.520,A 0.000,B 0.000,C 90.000,E1 273.669} C_DIS
LIN {X -0.022,Y -372.509,Z 1419.518,A 0.000,B 0.000,C 90.000,E1 273.212} C_DIS
LIN {X -0.101,Y -362.249,Z 1419.516,A 0.000,B 0.000,C 90.000,E1 272.922} C_DIS
LIN {X 0.130,Y -351.506,Z 1419.515,A 0.000,B 0.000,C 90.000,E1 272.636} C_DIS
LIN {X -0.037,Y -344.173,Z 1419.514,A 0.000,B 0.000,C 90.000,E1 272.522} C_DIS
LIN {X -0.062,Y -331.345,Z 1419.513,A 0.000,B 0.000,C 90.000,E1 272.350} C_DIS
LIN {X 0.048,Y -318.531,Z 1419.512,A 0.000,B 0.000,C 90.000,E1 272.236} C_DIS
LIN {X -0.100,Y -309.265,Z 1419.512,A 0.000,B 0.000,C 90.000,E1 272.236} C_DIS
LIN {X -0.088,Y -181.229,Z 1419.512,A 0.000,B 0.000,C 90.000,E1 272.236} C_DIS
LIN {X 0.091,Y -181.567,Z 1419.503,A 0.000,B 0.000,C 90.000,E1 270.458} C_DIS
LIN {X 0.080,Y -181.119,Z 1419.489,A 0.000,B 0.000,C 90.000,E1 267.936} C_DIS
LIN {X 0.068,Y -180.906,Z 1419.475,A 0.000,B 0.000,C 90.000,E1 265.412} C_DIS
LIN {X -0.056,Y -180.720,Z 1419.470,A 0.000,B 0.000,C 90.000,E1 264.609} C_DIS
LIN {X 0.042,Y -178.807,Z 1419.442,A 0.000,B 0.000,C 90.000,E1 259.511} C_DIS
LIN {X -0.051,Y -175.853,Z 1419.413,A 0.000,B 0.000,C 90.000,E1 254.448} C_DIS
LIN {X -0.069,Y -173.179,Z 1419.395,A 0.000,B 0.000,C 90.000,E1 251.040} C_DIS
LIN {X -0.066,Y -171.480,Z 1419.380,A 0.000,B 0.000,C 90.000,E1 248.465} C_DIS
LIN {X -0.079,Y -167.711,Z 1419.356,A 0.000,B 0.000,C 90.000,E1 244.152} C_DIS
LIN {X -0.062,Y -166.399,Z 1419.347,A 0.000,B 0.000,C 90.000,E1 242.410} C_DIS
LIN {X 0.077,Y -163.125,Z 1419.327,A 0.000,B 0.000,C 90.000,E1 238.869} C_DIS
LIN {X -0.097,Y -161.075,Z 1419.313,A 0.000,B 0.000,C 90.000,E1 236.294} C_DIS
LIN {X 0.013,Y -157.807,Z 1419.293,A 0.000,B 0.000,C 90.000,E1 232.718} C_DIS
LIN {X -0.048,Y -155.842,Z 1419.278,A 0.000,B 0.000,C 90.000,E1 230.070} C_DIS
LIN {X 0.008,Y -152.093,Z 1419.253,A 0.000,B 0.000,C 90.000,E1 225.567} C_DIS
LIN {X 0.027,Y -150.344,Z 1419.238,A 0.000,B 0.000,C 90.000,E1 222.852} C_DIS
LIN {X 0.047,Y -147.082,Z 1419.213,A 0.000,B 0.000,C 90.000,E1 218.302} C_DIS
LIN {X -0.049,Y -145.655,Z 1419.198,A 0.000,B 0.000,C 90.000,E1 215.598} C_DIS
LIN {X -0.045,Y -143.037,Z 1419.172,A 0.000,B 0.000,C 90.000,E1 211.003} C_DIS
LIN {X 0.081,Y -141.661,Z 1419.152,A 0.000,B 0.000,C 90.000,E1 207.257} C_DIS
LIN {X 0.000,Y -139.448,Z 1419.115,A 0.000,B 0.000,C 90.000,E1 200.791} C_DIS
LIN {X 0.053,Y -139.182,Z 1419.105,A 0.000,B 0.000,C 90.000,E1 198.906} C_DIS
LIN {X -0.055,Y -138.321,Z 1419.053,A 0.000,B 0.000,C 90.000,E1 189.613} C_DIS
LIN {X -0.049,Y -139.464,Z 1419.007,A 0.000,B 0.000,C 90.000,E1 181.203} C_DIS
LIN {X 0.031,Y -141.025,Z 1418.976,A 0.000,B 0.000,C 90.000,E1 175.584} C_DIS
LIN {X -0.013,Y -142.391,Z 1418.960,A 0.000,B 0.000,C 90.000,E1 172.818} C_DIS
LIN {X 0.049,Y -144.622,Z 1418.934,A 0.000,B 0.000,C 90.000,E1 168.173} C_DIS
LIN {X -0.032,Y -147.817,Z 1418.909,A 0.000,B 0.000,C 90.000,E1 163.614} C_DIS
LIN {X 0.055,Y -150.506,Z 1418.889,A 0.000,B 0.000,C 90.000,E1 159.934} C_DIS
LIN {X -0.066,Y -153.966,Z 1418.869,A 0.000,B 0.000,C 90.000,E1 156.357} C_DIS
LIN {X -0.003,Y -157.378,Z 1418.849,A 0.000,B 0.000,C 90.000,E1 152.743} C_DIS
LIN {X -0.062,Y -161.580,Z 1418.829,A 0.000,B 0.000,C 90.000,E1 149.203} C_DIS
LIN {X -0.050,Y -165.777,Z 1418.809,A 0.000,B 0.000,C 90.000,E1 145.674} C_DIS
LIN {X -0.065,Y -170.738,Z 1418.790,A 0.000,B 0.000,C 90.000,E1 142.190} C_DIS
LIN {X -0.022,Y -175.610,Z 1418.771,A 0.000,B 0.000,C 90.000,E1 138.728} C_DIS
LIN {X -0.036,Y -181.226,Z 1418.752,A 0.000,B 0.000,C 90.000,E1 135.324} C_DIS
LIN {X 0.095,Y -186.693,Z 1418.733,A 0.000,B 0.000,C 90.000,E1 131.919} C_DIS
LIN {X 0.047,Y -191.294,Z 1418.719,A 0.000,B 0.000,C 90.000,E1 129.439} C_DIS
LIN {X -0.021,Y -197.121,Z 1418.701,A 0.000,B 0.000,C 90.000,E1 126.171} C_DIS
LIN {X -0.101,Y -199.872,Z 1418.693,A 0.000,B 0.000,C 90.000,E1 124.818} C_DIS
LIN {X 0.056,Y -310.801,Z 1418.693,A 0.000,B 0.000,C 90.000,E1 124.771} C_DIS
LIN {X 0.015,Y -311.543,Z 1418.693,A 0.000,B 0.000,C 90.000,E1 124.771} C_DIS
LIN {X 0.023,Y -317.340,Z 1418.692,A 0.000,B 0.000,C 90.000,E1 124.532} C_DIS
LIN {X 0.012,Y -320.286,Z 1418.690,A 0.000,B 0.000,C 90.000,E1 124.278} C_DIS
LIN {X -0.031,Y -323.986,Z 1418.688,A 0.000,B 0.000,C 90.000,E1 123.785} C_DIS
LIN {X 0.053,Y -325.630,Z 1418.686,A 0.000,B 0.000,C 90.000,E1 123.452} C_DIS
LIN {X -0.036,Y -328.019,Z 1418.682,A 0.000,B 0.000,C 90.000,E1 122.832} C_DIS
LIN {X 0.023,Y -338.670,Z 1418.667,A 0.000,B 0.000,C 90.000,E1 120.001} C_DIS
LIN {X -0.125,Y -350.674,Z 1418.651,A 0.000,B 0.000,C 90.000,E1 117.257} C_DIS
LIN {X 0.058,Y -364.141,Z 1418.636,A 0.000,B 0.000,C 90.000,E1 114.515} C_DIS
LIN {X 0.077,Y -377.431,Z 1418.623,A 0.000,B 0.000,C 90.000,E1 112.153} C_DIS
LIN {X -0.073,Y -392.058,Z 1418.610,A 0.000,B 0.000,C 90.000,E1 109.866} C_DIS
LIN {X 0.113,Y -408.125,Z 1418.598,A 0.000,B 0.000,C 90.000,E1 107.583} C_DIS
LIN {X -0.204,Y -425.744,Z 1418.586,A 0.000,B 0.000,C 90.000,E1 105.426} C_DIS
LIN {X 0.136,Y -444.990,Z 1418.574,A 0.000,B 0.000,C 90.000,E1 103.244} C_DIS
LIN {X 0.225,Y -465.113,Z 1418.563,A 0.000,B 0.000,C 90.000,E1 101.243} C_DIS
LIN {X -0.025,Y -485.687,Z 1418.552,A 0.000,B 0.000,C 90.000,E1 99.443} C_DIS
LIN {X 0.068,Y -487.692,Z 1418.551,A 0.000,B 0.000,C 90.000,E1 99.208} C_DIS
LIN {X 0.160,Y -489.224,Z 1418.550,A 0.000,B 0.000,C 90.000,E1 98.973} C_DIS
LIN {X -0.016,Y -490.504,Z 1418.549,A 0.000,B 0.000,C 90.000,E1 98.746} C_DIS
LIN {X -0.118,Y -491.443,Z 1418.547,A 0.000,B 0.000,C 90.000,E1 98.511} C_DIS
LIN {X 0.106,Y -492.466,Z 1418.544,A 0.000,B 0.000,C 90.000,E1 97.992} C_DIS
LIN {X -0.149,Y -492.480,Z 1418.542,A 0.000,B 0.000,C 90.000,E1 97.530} C_DIS
LIN {X 0.091,Y -491.490,Z 1418.539,A 0.000,B 0.000,C 90.000,E1 97.011} C_DIS
LIN {X -0.005,Y -490.574,Z 1418.538,A 0.000,B 0.000,C 90.000,E1 96.777} C_DIS
LIN {X -0.101,Y -489.321,Z 1418.536,A 0.000,B 0.000,C 90.000,E1 96.543} C_DIS
LIN {X 0.105,Y -471.503,Z 1418.521,A 0.000,B 0.000,C 90.000,E1 93.784} C_DIS
LIN {X -0.182,Y -465.094,Z 1418.516,A 0.000,B 0.000,C 90.000,E1 92.808} C_DIS
LIN {X 0.169,Y -453.281,Z 1418.505,A 0.000,B 0.000,C 90.000,E1 90.974} C_DIS
LIN {X -0.082,Y -437.179,Z 1418.491,A 0.000,B 0.000,C 90.000,E1 88.396} C_DIS
LIN {X 0.017,Y -427.792,Z 1418.482,A 0.000,B 0.000,C 90.000,E1 86.788} C_DIS
LIN {X 0.058,Y -416.652,Z 1418.472,A 0.000,B 0.000,C 90.000,E1 84.894} C_DIS
LIN {X -0.097,Y -405.472,Z 1418.461,A 0.000,B 0.000,C 90.000,E1 82.996} C_DIS
LIN {X 0.010,Y -394.164,Z 1418.450,A 0.000,B 0.000,C 90.000,E1 81.027} C_DIS
LIN {X -0.050,Y -382.711,Z 1418.439,A 0.000,B 0.000,C 90.000,E1 79.050} C_DIS
LIN {X 0.172,Y -369.684,Z 1418.426,A 0.000,B 0.000,C 90.000,E1 76.700} C_DIS
LIN {X 0.201,Y -358.369,Z 1418.415,A 0.000,B 0.000,C 90.000,E1 74.629} C_DIS
LIN {X 0.089,Y -346.945,Z 1418.403,A 0.000,B 0.000,C 90.000,E1 72.543} C_DIS
LIN {X -0.052,Y -336.988,Z 1418.393,A 0.000,B 0.000,C 90.000,E1 70.732} C_DIS
LIN {X 0.018,Y -325.476,Z 1418.381,A 0.000,B 0.000,C 90.000,E1 68.539} C_DIS
LIN {X -0.108,Y -308.183,Z 1418.361,A 0.000,B 0.000,C 90.000,E1 65.049} C_DIS
LIN {X -0.143,Y -295.568,Z 1418.345,A 0.000,B 0.000,C 90.000,E1 62.103} C_DIS
LIN {X -0.098,Y -284.216,Z 1418.328,A 0.000,B 0.000,C 90.000,E1 59.076} C_DIS
LIN {X 0.156,Y -272.707,Z 1418.309,A 0.000,B 0.000,C 90.000,E1 55.595} C_DIS
LIN {X 0.092,Y -262.006,Z 1418.290,A 0.000,B 0.000,C 90.000,E1 52.110} C_DIS
LIN {X -0.013,Y -252.005,Z 1418.270,A 0.000,B 0.000,C 90.000,E1 48.566} C_DIS
LIN {X 0.035,Y -242.751,Z 1418.250,A 0.000,B 0.000,C 90.000,E1 44.919} C_DIS
LIN {X -0.019,Y -234.418,Z 1418.229,A 0.000,B 0.000,C 90.000,E1 41.229} C_DIS
LIN {X 0.067,Y -226.938,Z 1418.208,A 0.000,B 0.000,C 90.000,E1 37.443} C_DIS
LIN {X 0.043,Y -220.308,Z 1418.187,A 0.000,B 0.000,C 90.000,E1 33.627} C_DIS
LIN {X 0.069,Y -214.523,Z 1418.165,A 0.000,B 0.000,C 90.000,E1 29.745} C_DIS
LIN {X -0.019,Y -209.542,Z 1418.144,A 0.000,B 0.000,C 90.000,E1 25.848} C_DIS
LIN {X -0.058,Y -205.510,Z 1418.122,A 0.000,B 0.000,C 90.000,E1 21.897} C_DIS
LIN {X -0.038,Y -201.784,Z 1418.095,A 0.000,B 0.000,C 90.000,E1 17.094} C_DIS
LIN {X 0.024,Y -199.044,Z 1418.068,A 0.000,B 0.000,C 90.000,E1 12.243} C_DIS
LIN {X -0.070,Y -197.044,Z 1418.041,A 0.000,B 0.000,C 90.000,E1 7.409} C_DIS
LIN {X -0.012,Y -195.795,Z 1418.018,A 0.000,B 0.000,C 90.000,E1 3.326} C_DIS
LIN {X -0.084,Y -194.966,Z 1417.993,A 0.000,B 0.000,C 90.000,E1 358.740} C_DIS
LIN {X 0.006,Y -194.703,Z 1417.961,A 0.000,B 0.000,C 90.000,E1 352.996} C_DIS
LIN {X -0.017,Y -195.408,Z 1417.929,A 0.000,B 0.000,C 90.000,E1 347.285} C_DIS
LIN {X -0.077,Y -198.065,Z 1417.893,A 0.000,B 0.000,C 90.000,E1 340.786} C_DIS
LIN {X -0.051,Y -201.706,Z 1417.866,A 0.000,B 0.000,C 90.000,E1 335.921} C_DIS
LIN {X -0.021,Y -206.007,Z 1417.844,A 0.000,B 0.000,C 90.000,E1 331.897} C_DIS
LIN {X -0.001,Y -211.361,Z 1417.822,A 0.000,B 0.000,C 90.000,E1 327.916} C_DIS
LIN {X -0.001,Y -216.748,Z 1417.804,A 0.000,B 0.000,C 90.000,E1 324.769} C_DIS
LIN {X -0.015,Y -223.057,Z 1417.787,A 0.000,B 0.000,C 90.000,E1 321.662} C_DIS
LIN {X -0.075,Y -230.272,Z 1417.770,A 0.000,B 0.000,C 90.000,E1 318.609} C_DIS
LIN {X -0.015,Y -239.532,Z 1417.751,A 0.000,B 0.000,C 90.000,E1 315.202} C_DIS
LIN {X -0.027,Y -249.955,Z 1417.733,A 0.000,B 0.000,C 90.000,E1 311.881} C_DIS
LIN {X -0.053,Y -260.305,Z 1417.717,A 0.000,B 0.000,C 90.000,E1 308.991} C_DIS
LIN {X 0.033,Y -271.818,Z 1417.701,A 0.000,B 0.000,C 90.000,E1 306.137} C_DIS
LIN {X 0.045,Y -283.262,Z 1417.687,A 0.000,B 0.000,C 90.000,E1 303.706} C_DIS
LIN {X 0.056,Y -290.615,Z 1417.680,A 0.000,B 0.000,C 90.000,E1 302.339} C_DIS
LIN {X 0.006,Y -298.690,Z 1417.672,A 0.000,B 0.000,C 90.000,E1 301.003} C_DIS
LIN {X 0.059,Y -307.526,Z 1417.665,A 0.000,B 0.000,C 90.000,E1 299.667} C_DIS
LIN {X 0.017,Y -314.795,Z 1417.659,A 0.000,B 0.000,C 90.000,E1 298.693} C_DIS
LIN {X -0.006,Y -324.922,Z 1417.653,A 0.000,B 0.000,C 90.000,E1 297.462} C_DIS
LIN {X -0.007,Y -346.331,Z 1417.640,A 0.000,B 0.000,C 90.000,E1 295.155} C_DIS
LIN {X -0.066,Y -359.829,Z 1417.632,A 0.000,B 0.000,C 90.000,E1 293.770} C_DIS
LIN {X 0.086,Y -370.257,Z 1417.626,A 0.000,B 0.000,C 90.000,E1 292.642} C_DIS
LIN {X -0.017,Y -380.491,Z 1417.620,A 0.000,B 0.000,C 90.000,E1 291.535} C_DIS
LIN {X -0.076,Y -393.123,Z 1417.612,A 0.000,B 0.000,C 90.000,E1 290.120} C_DIS
LIN {X 0.029,Y -408.202,Z 1417.602,A 0.000,B 0.000,C 90.000,E1 288.417} C_DIS
LIN {X -0.029,Y -418.099,Z 1417.596,A 0.000,B 0.000,C 90.000,E1 287.330} C_DIS
LIN {X 0.079,Y -425.124,Z 1417.592,A 0.000,B 0.000,C 90.000,E1 286.496} C_DIS
LIN {X -0.164,Y -431.445,Z 1417.587,A 0.000,B 0.000,C 90.000,E1 285.717} C_DIS
LIN {X -0.045,Y -436.831,Z 1417.583,A 0.000,B 0.000,C 90.000,E1 284.898} C_DIS
LIN {X 0.034,Y -439.908,Z 1417.580,A 0.000,B 0.000,C 90.000,E1 284.356} C_DIS
LIN {X -0.193,Y -443.857,Z 1417.575,A 0.000,B 0.000,C 90.000,E1 283.592} C_DIS
LIN {X -0.179,Y -446.105,Z 1417.572,A 0.000,B 0.000,C 90.000,E1 283.063} C_DIS
LIN {X -0.149,Y -448.080,Z 1417.570,A 0.000,B 0.000,C 90.000,E1 282.535} C_DIS
LIN {X -0.113,Y -449.676,Z 1417.567,A 0.000,B 0.000,C 90.000,E1 282.007} C_DIS
LIN {X -0.065,Y -450.940,Z 1417.564,A 0.000,B 0.000,C 90.000,E1 281.478} C_DIS
LIN {X -0.010,Y -451.798,Z 1417.561,A 0.000,B 0.000,C 90.000,E1 280.950} C_DIS
LIN {X -0.031,Y -452.194,Z 1417.558,A 0.000,B 0.000,C 90.000,E1 280.433} C_DIS
LIN {X 0.037,Y -452.199,Z 1417.555,A 0.000,B 0.000,C 90.000,E1 279.905} C_DIS
LIN {X 0.103,Y -451.677,Z 1417.552,A 0.000,B 0.000,C 90.000,E1 279.378} C_DIS
LIN {X 0.095,Y -450.594,Z 1417.549,A 0.000,B 0.000,C 90.000,E1 278.859} C_DIS
LIN {X 0.087,Y -448.959,Z 1417.546,A 0.000,B 0.000,C 90.000,E1 278.341} C_DIS
LIN {X 0.136,Y -446.621,Z 1417.543,A 0.000,B 0.000,C 90.000,E1 277.814} C_DIS
LIN {X -0.129,Y -445.205,Z 1417.542,A 0.000,B 0.000,C 90.000,E1 277.587} C_DIS
LIN {X -0.161,Y -441.671,Z 1417.539,A 0.000,B 0.000,C 90.000,E1 277.068} C_DIS
LIN {X 0.064,Y -439.590,Z 1417.538,A 0.000,B 0.000,C 90.000,E1 276.777} C_DIS
LIN {X 0.002,Y -434.505,Z 1417.535,A 0.000,B 0.000,C 90.000,E1 276.258} C_DIS
LIN {X 0.053,Y -428.352,Z 1417.532,A 0.000,B 0.000,C 90.000,E1 275.739} C_DIS
LIN {X 0.193,Y -421.844,Z 1417.529,A 0.000,B 0.000,C 90.000,E1 275.277} C_DIS
LIN {X -0.038,Y -415.631,Z 1417.527,A 0.000,B 0.000,C 90.000,E1 274.935} C_DIS
LIN {X 0.170,Y -405.806,Z 1417.525,A 0.000,B 0.000,C 90.000,E1 274.416} C_DIS
LIN {X 0.073,Y -395.927,Z 1417.522,A 0.000,B 0.000,C 90.000,E1 274.012} C_DIS
LIN {X -0.141,Y -386.268,Z 1417.520,A 0.000,B 0.000,C 90.000,E1 273.669} C_DIS
LIN {X -0.172,Y -376.325,Z 1417.518,A 0.000,B 0.000,C 90.000,E1 273.326} C_DIS
LIN {X 0.081,Y -366.387,Z 1417.517,A 0.000,B 0.000,C 90.000,E1 272.980} C_DIS
LIN {X -0.173,Y -355.740,Z 1417.515,A 0.000,B 0.000,C 90.000,E1 272.751} C_DIS
LIN {X -0.095,Y -344.692,Z 1417.514,A 0.000,B 0.000,C 90.000,E1 272.522} C_DIS
LIN {X -0.120,Y -331.625,Z 1417.513,A 0.000,B 0.000,C 90.000,E1 272.350} C_DIS
LIN {X 0.005,Y -318.378,Z 1417.512,A 0.000,B 0.000,C 90.000,E1 272.236} C_DIS
LIN {X -0.092,Y -312.996,Z 1417.512,A 0.000,B 0.000,C 90.000,E1 272.236} C_DIS
LIN {X -0.081,Y -181.229,Z 1417.512,A 0.000,B 0.000,C 90.000,E1 272.236} C_DIS
LIN {X 0.072,Y -181.567,Z 1417.503,A 0.000,B 0.000,C 90.000,E1 270.458} C_DIS
LIN {X 0.061,Y -181.117,Z 1417.489,A 0.000,B 0.000,C 90.000,E1 267.936} C_DIS
LIN {X 0.049,Y -180.907,Z 1417.475,A 0.000,B 0.000,C 90.000,E1 265.412} C_DIS
LIN {X -0.074,Y -180.717,Z 1417.470,A 0.000,B 0.000,C 90.000,E1 264.609} C_DIS
LIN {X 0.023,Y -178.805,Z 1417.442,A 0.000,B 0.000,C 90.000,E1 259.511} C_DIS
LIN {X -0.070,Y -175.850,Z 1417.413,A 0.000,B 0.000,C 90.000,E1 254.448} C_DIS
LIN {X -0.103,Y -172.586,Z 1417.390,A 0.000,B 0.000,C 90.000,E1 250.188} C_DIS
LIN {X 0.075,Y -171.476,Z 1417.380,A 0.000,B 0.000,C 90.000,E1 248.411} C_DIS
LIN {X -0.096,Y -167.706,Z 1417.356,A 0.000,B 0.000,C 90.000,E1 244.152} C_DIS
LIN {X 0.068,Y -166.394,Z 1417.347,A 0.000,B 0.000,C 90.000,E1 242.359} C_DIS
LIN {X 0.059,Y -163.119,Z 1417.327,A 0.000,B 0.000,C 90.000,E1 238.869} C_DIS
LIN {X 0.019,Y -161.070,Z 1417.313,A 0.000,B 0.000,C 90.000,E1 236.246} C_DIS
LIN {X -0.004,Y -157.803,Z 1417.293,A 0.000,B 0.000,C 90.000,E1 232.718} C_DIS
LIN {X -0.065,Y -155.838,Z 1417.278,A 0.000,B 0.000,C 90.000,E1 230.070} C_DIS
LIN {X -0.009,Y -152.088,Z 1417.253,A 0.000,B 0.000,C 90.000,E1 225.567} C_DIS
LIN {X 0.010,Y -150.339,Z 1417.238,A 0.000,B 0.000,C 90.000,E1 222.852} C_DIS
LIN {X 0.031,Y -147.078,Z 1417.213,A 0.000,B 0.000,C 90.000,E1 218.302} C_DIS
LIN {X -0.065,Y -145.652,Z 1417.198,A 0.000,B 0.000,C 90.000,E1 215.598} C_DIS
LIN {X -0.061,Y -143.033,Z 1417.172,A 0.000,B 0.000,C 90.000,E1 211.003} C_DIS
LIN {X 0.065,Y -141.658,Z 1417.152,A 0.000,B 0.000,C 90.000,E1 207.257} C_DIS
LIN {X -0.015,Y -139.447,Z 1417.115,A 0.000,B 0.000,C 90.000,E1 200.791} C_DIS
LIN {X 0.037,Y -139.181,Z 1417.105,A 0.000,B 0.000,C 90.000,E1 198.906} C_DIS
LIN {X 0.065,Y -138.320,Z 1417.053,A 0.000,B 0.000,C 90.000,E1 189.557} C_DIS
LIN {X -0.064,Y -139.465,Z 1417.007,A 0.000,B 0.000,C 90.000,E1 181.203} C_DIS
LIN {X 0.016,Y -141.029,Z 1416.975,A 0.000,B 0.000,C 90.000,E1 175.584} C_DIS
LIN {X -0.030,Y -142.394,Z 1416.960,A 0.000,B 0.000,C 90.000,E1 172.818} C_DIS
LIN {X 0.032,Y -144.626,Z 1416.934,A 0.000,B 0.000,C 90.000,E1 168.173} C_DIS
LIN {X -0.049,Y -147.821,Z 1416.909,A 0.000,B 0.000,C 90.000,E1 163.614} C_DIS
LIN {X 0.038,Y -150.513,Z 1416.889,A 0.000,B 0.000,C 90.000,E1 159.934} C_DIS
LIN {X 0.059,Y -153.973,Z 1416.869,A 0.000,B 0.000,C 90.000,E1 156.305} C_DIS
LIN {X -0.021,Y -157.385,Z 1416.849,A 0.000,B 0.000,C 90.000,E1 152.743} C_DIS
LIN {X -0.079,Y -161.588,Z 1416.829,A 0.000,B 0.000,C 90.000,E1 149.203} C_DIS
LIN {X -0.067,Y -165.785,Z 1416.809,A 0.000,B 0.000,C 90.000,E1 145.674} C_DIS
LIN {X -0.083,Y -170.747,Z 1416.790,A 0.000,B 0.000,C 90.000,E1 142.190} C_DIS
LIN {X 0.075,Y -175.619,Z 1416.771,A 0.000,B 0.000,C 90.000,E1 138.690} C_DIS
LIN {X -0.055,Y -181.235,Z 1416.752,A 0.000,B 0.000,C 90.000,E1 135.324} C_DIS
LIN {X 0.077,Y -186.704,Z 1416.733,A 0.000,B 0.000,C 90.000,E1 131.919} C_DIS
LIN {X 0.028,Y -191.303,Z 1416.719,A 0.000,B 0.000,C 90.000,E1 129.439} C_DIS
LIN {X -0.041,Y -197.133,Z 1416.701,A 0.000,B 0.000,C 90.000,E1 126.171} C_DIS
LIN {X -0.034,Y -199.832,Z 1416.693,A 0.000,B 0.000,C 90.000,E1 124.818} C_DIS
LIN {X -0.100,Y -310.969,Z 1416.693,A 0.000,B 0.000,C 90.000,E1 124.818} C_DIS
LIN {X -0.145,Y -315.448,Z 1416.693,A 0.000,B 0.000,C 90.000,E1 124.692} C_DIS
LIN {X -0.008,Y -317.609,Z 1416.692,A 0.000,B 0.000,C 90.000,E1 124.532} C_DIS
LIN {X 0.195,Y -321.477,Z 1416.690,A 0.000,B 0.000,C 90.000,E1 124.119} C_DIS
LIN {X 0.153,Y -324.945,Z 1416.687,A 0.000,B 0.000,C 90.000,E1 123.579} C_DIS
LIN {X -0.031,Y -326.357,Z 1416.685,A 0.000,B 0.000,C 90.000,E1 123.293} C_DIS
LIN {X 0.102,Y -338.078,Z 1416.667,A 0.000,B 0.000,C 90.000,E1 120.129} C_DIS
LIN {X -0.065,Y -350.014,Z 1416.652,A 0.000,B 0.000,C 90.000,E1 117.385} C_DIS
LIN {X 0.105,Y -363.401,Z 1416.637,A 0.000,B 0.000,C 90.000,E1 114.643} C_DIS
LIN {X 0.109,Y -376.618,Z 1416.624,A 0.000,B 0.000,C 90.000,E1 112.280} C_DIS
LIN {X -0.057,Y -391.166,Z 1416.611,A 0.000,B 0.000,C 90.000,E1 109.993} C_DIS
LIN {X 0.236,Y -407.148,Z 1416.599,A 0.000,B 0.000,C 90.000,E1 107.692} C_DIS
LIN {X -0.108,Y -424.675,Z 1416.586,A 0.000,B 0.000,C 90.000,E1 105.536} C_DIS
LIN {X 0.187,Y -443.837,Z 1416.574,A 0.000,B 0.000,C 90.000,E1 103.355} C_DIS
LIN {X 0.101,Y -463.928,Z 1416.563,A 0.000,B 0.000,C 90.000,E1 101.366} C_DIS
LIN {X -0.139,Y -484.554,Z 1416.553,A 0.000,B 0.000,C 90.000,E1 99.557} C_DIS
LIN {X -0.011,Y -486.774,Z 1416.552,A 0.000,B 0.000,C 90.000,E1 99.321} C_DIS
LIN {X -0.154,Y -488.604,Z 1416.550,A 0.000,B 0.000,C 90.000,E1 99.095} C_DIS
LIN {X -0.218,Y -489.984,Z 1416.549,A 0.000,B 0.000,C 90.000,E1 98.859} C_DIS
LIN {X -0.006,Y -491.761,Z 1416.546,A 0.000,B 0.000,C 90.000,E1 98.341} C_DIS
LIN {X -0.202,Y -492.434,Z 1416.544,A 0.000,B 0.000,C 90.000,E1 97.871} C_DIS
LIN {X 0.030,Y -492.114,Z 1416.541,A 0.000,B 0.000,C 90.000,E1 97.352} C_DIS
LIN {X -0.221,Y -490.757,Z 1416.538,A 0.000,B 0.000,C 90.000,E1 96.891} C_DIS
LIN {X 0.111,Y -489.620,Z 1416.537,A 0.000,B 0.000,C 90.000,E1 96.606} C_DIS
LIN {X -0.145,Y -486.374,Z 1416.534,A 0.000,B 0.000,C 90.000,E1 96.144} C_DIS
LIN {X -0.007,Y -468.704,Z 1416.519,A 0.000,B 0.000,C 90.000,E1 93.383} C_DIS
LIN {X -0.069,Y -460.439,Z 1416.512,A 0.000,B 0.000,C 90.000,E1 92.121} C_DIS
LIN {X 0.016,Y -439.094,Z 1416.493,A 0.000,B 0.000,C 90.000,E1 88.740} C_DIS
LIN {X 0.125,Y -429.812,Z 1416.484,A 0.000,B 0.000,C 90.000,E1 87.135} C_DIS
LIN {X -0.219,Y -418.721,Z 1416.474,A 0.000,B 0.000,C 90.000,E1 85.298} C_DIS
LIN {X 0.180,Y -405.964,Z 1416.462,A 0.000,B 0.000,C 90.000,E1 83.053} C_DIS
LIN {X -0.173,Y -396.300,Z 1416.452,A 0.000,B 0.000,C 90.000,E1 81.432} C_DIS
LIN {X -0.182,Y -384.904,Z 1416.441,A 0.000,B 0.000,C 90.000,E1 79.454} C_DIS
LIN {X 0.020,Y -371.850,Z 1416.428,A 0.000,B 0.000,C 90.000,E1 77.117} C_DIS
LIN {X 0.096,Y -360.541,Z 1416.417,A 0.000,B 0.000,C 90.000,E1 75.046} C_DIS
LIN {X 0.032,Y -349.119,Z 1416.405,A 0.000,B 0.000,C 90.000,E1 72.960} C_DIS
LIN {X -0.065,Y -339.189,Z 1416.395,A 0.000,B 0.000,C 90.000,E1 71.148} C_DIS
LIN {X 0.032,Y -325.992,Z 1416.381,A 0.000,B 0.000,C 90.000,E1 68.646} C_DIS
LIN {X -0.069,Y -308.635,Z 1416.362,A 0.000,B 0.000,C 90.000,E1 65.153} C_DIS
LIN {X -0.091,Y -297.325,Z 1416.347,A 0.000,B 0.000,C 90.000,E1 62.538} C_DIS
LIN {X -0.134,Y -285.803,Z 1416.331,A 0.000,B 0.000,C 90.000,E1 59.537} C_DIS
LIN {X 0.023,Y -274.191,Z 1416.312,A 0.000,B 0.000,C 90.000,E1 56.087} C_DIS
LIN {X 0.002,Y -263.449,Z 1416.292,A 0.000,B 0.000,C 90.000,E1 52.603} C_DIS
LIN {X -0.046,Y -253.346,Z 1416.272,A 0.000,B 0.000,C 90.000,E1 49.057} C_DIS
LIN {X 0.069,Y -245.845,Z 1416.256,A 0.000,B 0.000,C 90.000,E1 46.134} C_DIS
LIN {X 0.095,Y -237.192,Z 1416.236,A 0.000,B 0.000,C 90.000,E1 42.447} C_DIS
LIN {X -0.092,Y -229.481,Z 1416.215,A 0.000,B 0.000,C 90.000,E1 38.749} C_DIS
LIN {X 0.100,Y -222.585,Z 1416.194,A 0.000,B 0.000,C 90.000,E1 34.898} C_DIS
LIN {X 0.058,Y -216.524,Z 1416.173,A 0.000,B 0.000,C 90.000,E1 31.052} C_DIS
LIN {X -0.062,Y -211.292,Z 1416.151,A 0.000,B 0.000,C 90.000,E1 27.180} C_DIS
LIN {X 0.034,Y -206.962,Z 1416.129,A 0.000,B 0.000,C 90.000,E1 23.206} C_DIS
LIN {X 0.057,Y -202.978,Z 1416.102,A 0.000,B 0.000,C 90.000,E1 18.417} C_DIS
LIN {X 0.068,Y -200.025,Z 1416.076,A 0.000,B 0.000,C 90.000,E1 13.592} C_DIS
LIN {X 0.049,Y -197.883,Z 1416.049,A 0.000,B 0.000,C 90.000,E1 8.746} C_DIS
LIN {X -0.002,Y -196.521,Z 1416.026,A 0.000,B 0.000,C 90.000,E1 4.702} C_DIS
LIN {X -0.035,Y -195.374,Z 1415.997,A 0.000,B 0.000,C 90.000,E1 359.542} C_DIS
LIN {X 0.089,Y -194.947,Z 1415.970,A 0.000,B 0.000,C 90.000,E1 354.609} C_DIS
LIN {X -0.038,Y -195.229,Z 1415.943,A 0.000,B 0.000,C 90.000,E1 349.746} C_DIS
LIN {X -0.059,Y -197.453,Z 1415.902,A 0.000,B 0.000,C 90.000,E1 342.417} C_DIS
LIN {X -0.015,Y -200.536,Z 1415.875,A 0.000,B 0.000,C 90.000,E1 337.539} C_DIS
LIN {X -0.013,Y -204.377,Z 1415.853,A 0.000,B 0.000,C 90.000,E1 333.512} C_DIS
LIN {X -0.072,Y -209.260,Z 1415.831,A 0.000,B 0.000,C 90.000,E1 329.537} C_DIS
LIN {X 0.054,Y -214.140,Z 1415.813,A 0.000,B 0.000,C 90.000,E1 326.342} C_DIS
LIN {X 0.069,Y -219.994,Z 1415.796,A 0.000,B 0.000,C 90.000,E1 323.210} C_DIS
LIN {X -0.041,Y -226.738,Z 1415.779,A 0.000,B 0.000,C 90.000,E1 320.150} C_DIS
LIN {X 0.075,Y -235.432,Z 1415.760,A 0.000,B 0.000,C 90.000,E1 316.701} C_DIS
LIN {X -0.055,Y -245.346,Z 1415.741,A 0.000,B 0.000,C 90.000,E1 313.380} C_DIS
LIN {X -0.038,Y -256.405,Z 1415.723,A 0.000,B 0.000,C 90.000,E1 310.092} C_DIS
LIN {X 0.009,Y -268.925,Z 1415.705,A 0.000,B 0.000,C 90.000,E1 306.870} C_DIS
LIN {X 0.016,Y -278.278,Z 1415.693,A 0.000,B 0.000,C 90.000,E1 304.771} C_DIS
LIN {X 0.089,Y -286.912,Z 1415.684,A 0.000,B 0.000,C 90.000,E1 303.038} C_DIS
LIN {X 0.140,Y -296.620,Z 1415.674,A 0.000,B 0.000,C 90.000,E1 301.337} C_DIS
LIN {X 0.170,Y -305.251,Z 1415.667,A 0.000,B 0.000,C 90.000,E1 300.001} C_DIS
LIN {X -0.117,Y -314.800,Z 1415.660,A 0.000,B 0.000,C 90.000,E1 298.743} C_DIS
LIN {X 0.138,Y -327.880,Z 1415.651,A 0.000,B 0.000,C 90.000,E1 297.129} C_DIS
LIN {X 0.078,Y -346.892,Z 1415.640,A 0.000,B 0.000,C 90.000,E1 295.103} C_DIS
LIN {X 0.086,Y -360.272,Z 1415.632,A 0.000,B 0.000,C 90.000,E1 293.718} C_DIS
LIN {X 0.152,Y -370.805,Z 1415.626,A 0.000,B 0.000,C 90.000,E1 292.589} C_DIS
LIN {X 0.103,Y -381.136,Z 1415.619,A 0.000,B 0.000,C 90.000,E1 291.461} C_DIS
LIN {X -0.160,Y -393.829,Z 1415.611,A 0.000,B 0.000,C 90.000,E1 290.066} C_DIS
LIN {X -0.060,Y -411.230,Z 1415.601,A 0.000,B 0.000,C 90.000,E1 288.109} C_DIS
LIN {X 0.153,Y -421.019,Z 1415.594,A 0.000,B 0.000,C 90.000,E1 286.985} C_DIS
LIN {X -0.122,Y -427.805,Z 1415.590,A 0.000,B 0.000,C 90.000,E1 286.205} C_DIS
LIN {X -0.095,Y -431.886,Z 1415.587,A 0.000,B 0.000,C 90.000,E1 285.662} C_DIS
LIN {X -0.160,Y -435.556,Z 1415.584,A 0.000,B 0.000,C 90.000,E1 285.134} C_DIS
LIN {X 0.115,Y -440.298,Z 1415.580,A 0.000,B 0.000,C 90.000,E1 284.300} C_DIS
LIN {X -0.106,Y -444.245,Z 1415.575,A 0.000,B 0.000,C 90.000,E1 283.536} C_DIS
LIN {X -0.088,Y -446.500,Z 1415.572,A 0.000,B 0.000,C 90.000,E1 283.008} C_DIS
LIN {X -0.055,Y -448.452,Z 1415.569,A 0.000,B 0.000,C 90.000,E1 282.479} C_DIS
LIN {X -0.015,Y -450.046,Z 1415.566,A 0.000,B 0.000,C 90.000,E1 281.951} C_DIS
LIN {X 0.035,Y -451.281,Z 1415.563,A 0.000,B 0.000,C 90.000,E1 281.422} C_DIS
LIN {X 0.094,Y -452.087,Z 1415.561,A 0.000,B 0.000,C 90.000,E1 280.894} C_DIS
LIN {X 0.158,Y -452.505,Z 1415.558,A 0.000,B 0.000,C 90.000,E1 280.366} C_DIS
LIN {X 0.147,Y -452.461,Z 1415.555,A 0.000,B 0.000,C 90.000,E1 279.849} C_DIS
LIN {X 0.214,Y -451.943,Z 1415.552,A 0.000,B 0.000,C 90.000,E1 279.321} C_DIS
LIN {X 0.209,Y -450.819,Z 1415.549,A 0.000,B 0.000,C 90.000,E1 278.803} C_DIS
LIN {X -0.177,Y -449.127,Z 1415.546,A 0.000,B 0.000,C 90.000,E1 278.333} C_DIS
LIN {X -0.189,Y -446.788,Z 1415.543,A 0.000,B 0.000,C 90.000,E1 277.814} C_DIS
LIN {X -0.011,Y -445.339,Z 1415.542,A 0.000,B 0.000,C 90.000,E1 277.530} C_DIS
LIN {X 0.011,Y -441.757,Z 1415.539,A 0.000,B 0.000,C 90.000,E1 277.004} C_DIS
LIN {X 0.182,Y -439.688,Z 1415.537,A 0.000,B 0.000,C 90.000,E1 276.720} C_DIS
LIN {X 0.119,Y -434.543,Z 1415.535,A 0.000,B 0.000,C 90.000,E1 276.201} C_DIS
LIN {X -0.171,Y -428.520,Z 1415.532,A 0.000,B 0.000,C 90.000,E1 275.739} C_DIS
LIN {X -0.002,Y -422.090,Z 1415.529,A 0.000,B 0.000,C 90.000,E1 275.277} C_DIS
LIN {X 0.174,Y -415.840,Z 1415.527,A 0.000,B 0.000,C 90.000,E1 274.878} C_DIS
LIN {X -0.170,Y -409.284,Z 1415.525,A 0.000,B 0.000,C 90.000,E1 274.588} C_DIS
LIN {X -0.054,Y -399.294,Z 1415.523,A 0.000,B 0.000,C 90.000,E1 274.131} C_DIS
LIN {X 0.024,Y -386.374,Z 1415.520,A 0.000,B 0.000,C 90.000,E1 273.612} C_DIS
LIN {X -0.008,Y -376.429,Z 1415.518,A 0.000,B 0.000,C 90.000,E1 273.269} C_DIS
LIN {X -0.114,Y -366.317,Z 1415.516,A 0.000,B 0.000,C 90.000,E1 272.980} C_DIS
LIN {X 0.068,Y -355.990,Z 1415.515,A 0.000,B 0.000,C 90.000,E1 272.694} C_DIS
LIN {X -0.165,Y -345.237,Z 1415.514,A 0.000,B 0.000,C 90.000,E1 272.522} C_DIS
LIN {X 0.147,Y -336.889,Z 1415.513,A 0.000,B 0.000,C 90.000,E1 272.350} C_DIS
LIN {X 0.099,Y -322.840,Z 1415.513,A 0.000,B 0.000,C 90.000,E1 272.236} C_DIS
LIN {X -0.118,Y -312.622,Z 1415.512,A 0.000,B 0.000,C 90.000,E1 272.236} C_DIS
LIN {X 0.085,Y -181.229,Z 1415.512,A 0.000,B 0.000,C 90.000,E1 272.178} C_DIS
LIN {X 0.064,Y -181.568,Z 1415.503,A 0.000,B 0.000,C 90.000,E1 270.458} C_DIS
LIN {X 0.053,Y -181.117,Z 1415.489,A 0.000,B 0.000,C 90.000,E1 267.936} C_DIS
LIN {X 0.041,Y -180.906,Z 1415.475,A 0.000,B 0.000,C 90.000,E1 265.412} C_DIS
LIN {X -0.082,Y -180.716,Z 1415.470,A 0.000,B 0.000,C 90.000,E1 264.609} C_DIS
LIN {X 0.016,Y -178.803,Z 1415.442,A 0.000,B 0.000,C 90.000,E1 259.511} C_DIS
LIN {X 0.092,Y -175.849,Z 1415.413,A 0.000,B 0.000,C 90.000,E1 254.393} C_DIS
LIN {X 0.052,Y -172.584,Z 1415.390,A 0.000,B 0.000,C 90.000,E1 250.134} C_DIS
LIN {X 0.068,Y -171.473,Z 1415.380,A 0.000,B 0.000,C 90.000,E1 248.411} C_DIS
LIN {X 0.047,Y -167.704,Z 1415.356,A 0.000,B 0.000,C 90.000,E1 244.101} C_DIS
LIN {X 0.060,Y -166.391,Z 1415.347,A 0.000,B 0.000,C 90.000,E1 242.359} C_DIS
LIN {X 0.052,Y -163.117,Z 1415.327,A 0.000,B 0.000,C 90.000,E1 238.869} C_DIS
LIN {X 0.102,Y -161.066,Z 1415.313,A 0.000,B 0.000,C 90.000,E1 236.215} C_DIS
LIN {X -0.012,Y -157.800,Z 1415.293,A 0.000,B 0.000,C 90.000,E1 232.718} C_DIS
LIN {X -0.073,Y -155.836,Z 1415.278,A 0.000,B 0.000,C 90.000,E1 230.070} C_DIS
LIN {X -0.017,Y -152.086,Z 1415.253,A 0.000,B 0.000,C 90.000,E1 225.567} C_DIS
LIN {X 0.003,Y -150.337,Z 1415.238,A 0.000,B 0.000,C 90.000,E1 222.852} C_DIS
LIN {X 0.023,Y -147.076,Z 1415.213,A 0.000,B 0.000,C 90.000,E1 218.302} C_DIS
LIN {X -0.073,Y -145.650,Z 1415.198,A 0.000,B 0.000,C 90.000,E1 215.598} C_DIS
LIN {X -0.068,Y -143.032,Z 1415.172,A 0.000,B 0.000,C 90.000,E1 211.003} C_DIS
LIN {X 0.058,Y -141.657,Z 1415.152,A 0.000,B 0.000,C 90.000,E1 207.257} C_DIS
LIN {X -0.023,Y -139.446,Z 1415.115,A 0.000,B 0.000,C 90.000,E1 200.791} C_DIS
LIN {X 0.030,Y -139.179,Z 1415.105,A 0.000,B 0.000,C 90.000,E1 198.906} C_DIS
LIN {X 0.058,Y -138.320,Z 1415.053,A 0.000,B 0.000,C 90.000,E1 189.557} C_DIS
LIN {X 0.068,Y -139.465,Z 1415.006,A 0.000,B 0.000,C 90.000,E1 181.146} C_DIS
LIN {X 0.009,Y -141.029,Z 1414.975,A 0.000,B 0.000,C 90.000,E1 175.584} C_DIS
LIN {X -0.037,Y -142.396,Z 1414.960,A 0.000,B 0.000,C 90.000,E1 172.818} C_DIS
LIN {X 0.025,Y -144.628,Z 1414.934,A 0.000,B 0.000,C 90.000,E1 168.173} C_DIS
LIN {X -0.056,Y -147.823,Z 1414.909,A 0.000,B 0.000,C 90.000,E1 163.614} C_DIS
LIN {X 0.031,Y -150.514,Z 1414.889,A 0.000,B 0.000,C 90.000,E1 159.934} C_DIS
LIN {X 0.051,Y -153.976,Z 1414.868,A 0.000,B 0.000,C 90.000,E1 156.305} C_DIS
LIN {X -0.028,Y -157.388,Z 1414.849,A 0.000,B 0.000,C 90.000,E1 152.743} C_DIS
LIN {X -0.086,Y -161.591,Z 1414.829,A 0.000,B 0.000,C 90.000,E1 149.203} C_DIS
LIN {X -0.076,Y -165.788,Z 1414.809,A 0.000,B 0.000,C 90.000,E1 145.674} C_DIS
LIN {X -0.090,Y -170.751,Z 1414.790,A 0.000,B 0.000,C 90.000,E1 142.190} C_DIS
LIN {X 0.068,Y -175.623,Z 1414.771,A 0.000,B 0.000,C 90.000,E1 138.690} C_DIS
LIN {X -0.062,Y -181.238,Z 1414.752,A 0.000,B 0.000,C 90.000,E1 135.324} C_DIS
LIN {X 0.068,Y -186.708,Z 1414.733,A 0.000,B 0.000,C 90.000,E1 131.919} C_DIS
LIN {X 0.019,Y -191.308,Z 1414.719,A 0.000,B 0.000,C 90.000,E1 129.439} C_DIS
LIN {X -0.050,Y -197.137,Z 1414.701,A 0.000,B 0.000,C 90.000,E1 126.171} C_DIS
LIN {X 0.051,Y -199.782,Z 1414.693,A 0.000,B 0.000,C 90.000,E1 124.818} C_DIS
LIN {X 0.032,Y -310.312,Z 1414.693,A 0.000,B 0.000,C 90.000,E1 124.818} C_DIS
LIN {X -0.110,Y -312.288,Z 1414.693,A 0.000,B 0.000,C 90.000,E1 124.818} C_DIS
LIN {X -0.022,Y -317.823,Z 1414.692,A 0.000,B 0.000,C 90.000,E1 124.532} C_DIS
LIN {X 0.159,Y -320.949,Z 1414.690,A 0.000,B 0.000,C 90.000,E1 124.199} C_DIS
LIN {X -0.127,Y -324.560,Z 1414.687,A 0.000,B 0.000,C 90.000,E1 123.706} C_DIS
LIN {X -0.042,Y -326.037,Z 1414.685,A 0.000,B 0.000,C 90.000,E1 123.372} C_DIS
LIN {X -0.071,Y -339.007,Z 1414.666,A 0.000,B 0.000,C 90.000,E1 119.922} C_DIS
LIN {X 0.095,Y -351.058,Z 1414.651,A 0.000,B 0.000,C 90.000,E1 117.129} C_DIS
LIN {X -0.186,Y -364.576,Z 1414.636,A 0.000,B 0.000,C 90.000,E1 114.463} C_DIS
LIN {X -0.016,Y -377.914,Z 1414.623,A 0.000,B 0.000,C 90.000,E1 112.078} C_DIS
LIN {X 0.069,Y -392.595,Z 1414.610,A 0.000,B 0.000,C 90.000,E1 109.758} C_DIS
LIN {X 0.019,Y -408.717,Z 1414.597,A 0.000,B 0.000,C 90.000,E1 107.511} C_DIS
LIN {X -0.001,Y -426.398,Z 1414.585,A 0.000,B 0.000,C 90.000,E1 105.315} C_DIS
LIN {X 0.050,Y -445.699,Z 1414.573,A 0.000,B 0.000,C 90.000,E1 103.175} C_DIS
LIN {X 0.083,Y -465.843,Z 1414.562,A 0.000,B 0.000,C 90.000,E1 101.186} C_DIS
LIN {X -0.166,Y -483.894,Z 1414.553,A 0.000,B 0.000,C 90.000,E1 99.613} C_DIS
LIN {X -0.043,Y -486.245,Z 1414.552,A 0.000,B 0.000,C 90.000,E1 99.378} C_DIS
LIN {X -0.121,Y -488.120,Z 1414.551,A 0.000,B 0.000,C 90.000,E1 99.151} C_DIS
LIN {X -0.120,Y -489.543,Z 1414.549,A 0.000,B 0.000,C 90.000,E1 98.916} C_DIS
LIN {X 0.089,Y -491.469,Z 1414.547,A 0.000,B 0.000,C 90.000,E1 98.398} C_DIS
LIN {X -0.177,Y -492.263,Z 1414.544,A 0.000,B 0.000,C 90.000,E1 97.936} C_DIS
LIN {X 0.121,Y -492.061,Z 1414.541,A 0.000,B 0.000,C 90.000,E1 97.409} C_DIS
LIN {X -0.133,Y -490.836,Z 1414.538,A 0.000,B 0.000,C 90.000,E1 96.947} C_DIS
LIN {X 0.199,Y -489.779,Z 1414.537,A 0.000,B 0.000,C 90.000,E1 96.663} C_DIS
LIN {X 0.101,Y -488.356,Z 1414.536,A 0.000,B 0.000,C 90.000,E1 96.429} C_DIS
LIN {X 0.145,Y -473.614,Z 1414.523,A 0.000,B 0.000,C 90.000,E1 94.188} C_DIS
LIN {X 0.179,Y -465.687,Z 1414.516,A 0.000,B 0.000,C 90.000,E1 92.922} C_DIS
LIN {X -0.153,Y -455.603,Z 1414.508,A 0.000,B 0.000,C 90.000,E1 91.432} C_DIS
LIN {X -0.155,Y -437.795,Z 1414.492,A 0.000,B 0.000,C 90.000,E1 88.568} C_DIS
LIN {X -0.066,Y -428.505,Z 1414.483,A 0.000,B 0.000,C 90.000,E1 86.963} C_DIS
LIN {X 0.023,Y -417.445,Z 1414.473,A 0.000,B 0.000,C 90.000,E1 85.065} C_DIS
LIN {X -0.115,Y -406.314,Z 1414.462,A 0.000,B 0.000,C 90.000,E1 83.166} C_DIS
LIN {X 0.020,Y -395.066,Z 1414.451,A 0.000,B 0.000,C 90.000,E1 81.197} C_DIS
LIN {X -0.020,Y -383.669,Z 1414.440,A 0.000,B 0.000,C 90.000,E1 79.218} C_DIS
LIN {X 0.148,Y -370.621,Z 1414.427,A 0.000,B 0.000,C 90.000,E1 76.881} C_DIS
LIN {X -0.147,Y -359.318,Z 1414.416,A 0.000,B 0.000,C 90.000,E1 74.866} C_DIS
LIN {X 0.100,Y -347.859,Z 1414.404,A 0.000,B 0.000,C 90.000,E1 72.725} C_DIS
LIN {X -0.024,Y -337.918,Z 1414.394,A 0.000,B 0.000,C 90.000,E1 70.913} C_DIS
LIN {X 0.034,Y -324.706,Z 1414.380,A 0.000,B 0.000,C 90.000,E1 68.411} C_DIS
LIN {X -0.116,Y -307.477,Z 1414.361,A 0.000,B 0.000,C 90.000,E1 64.921} C_DIS
LIN {X -0.030,Y -294.938,Z 1414.344,A 0.000,B 0.000,C 90.000,E1 61.948} C_DIS
LIN {X -0.024,Y -282.493,Z 1414.325,A 0.000,B 0.000,C 90.000,E1 58.584} C_DIS
LIN {X 0.027,Y -271.158,Z 1414.306,A 0.000,B 0.000,C 90.000,E1 55.135} C_DIS
LIN {X 0.015,Y -261.672,Z 1414.289,A 0.000,B 0.000,C 90.000,E1 51.984} C_DIS
LIN {X 0.062,Y -251.738,Z 1414.269,A 0.000,B 0.000,C 90.000,E1 48.405} C_DIS
LIN {X 0.101,Y -242.554,Z 1414.249,A 0.000,B 0.000,C 90.000,E1 44.757} C_DIS
LIN {X 0.038,Y -234.318,Z 1414.228,A 0.000,B 0.000,C 90.000,E1 41.067} C_DIS
LIN {X -0.023,Y -226.913,Z 1414.207,A 0.000,B 0.000,C 90.000,E1 37.317} C_DIS
LIN {X -0.039,Y -220.332,Z 1414.186,A 0.000,B 0.000,C 90.000,E1 33.499} C_DIS
LIN {X -0.006,Y -214.640,Z 1414.165,A 0.000,B 0.000,C 90.000,E1 29.617} C_DIS
LIN {X -0.089,Y -209.737,Z 1414.143,A 0.000,B 0.000,C 90.000,E1 25.720} C_DIS
LIN {X 0.076,Y -205.167,Z 1414.116,A 0.000,B 0.000,C 90.000,E1 20.918} C_DIS
LIN {X 0.073,Y -201.273,Z 1414.085,A 0.000,B 0.000,C 90.000,E1 15.315} C_DIS
LIN {X 0.029,Y -198.879,Z 1414.058,A 0.000,B 0.000,C 90.000,E1 10.489} C_DIS
LIN {X 0.065,Y -197.375,Z 1414.036,A 0.000,B 0.000,C 90.000,E1 6.429} C_DIS
LIN {X -0.079,Y -196.206,Z 1414.013,A 0.000,B 0.000,C 90.000,E1 2.407} C_DIS
LIN {X 0.074,Y -195.433,Z 1413.988,A 0.000,B 0.000,C 90.000,E1 357.879} C_DIS
LIN {X 0.034,Y -195.220,Z 1413.961,A 0.000,B 0.000,C 90.000,E1 352.996} C_DIS
LIN {X -0.009,Y -195.929,Z 1413.929,A 0.000,B 0.000,C 90.000,E1 347.297} C_DIS
LIN {X 0.001,Y -198.543,Z 1413.893,A 0.000,B 0.000,C 90.000,E1 340.786} C_DIS
LIN {X 0.045,Y -202.164,Z 1413.866,A 0.000,B 0.000,C 90.000,E1 335.921} C_DIS
LIN {X 0.092,Y -206.457,Z 1413.844,A 0.000,B 0.000,C 90.000,E1 331.897} C_DIS
LIN {X 0.016,Y -211.789,Z 1413.822,A 0.000,B 0.000,C 90.000,E1 327.946} C_DIS
LIN {X -0.034,Y -217.156,Z 1413.804,A 0.000,B 0.000,C 90.000,E1 324.815} C_DIS
LIN {X 0.005,Y -223.448,Z 1413.787,A 0.000,B 0.000,C 90.000,E1 321.698} C_DIS
LIN {X 0.099,Y -230.638,Z 1413.770,A 0.000,B 0.000,C 90.000,E1 318.609} C_DIS
LIN {X 0.005,Y -239.849,Z 1413.751,A 0.000,B 0.000,C 90.000,E1 315.243} C_DIS
LIN {X 0.014,Y -250.218,Z 1413.733,A 0.000,B 0.000,C 90.000,E1 311.919} C_DIS
LIN {X -0.032,Y -260.559,Z 1413.717,A 0.000,B 0.000,C 90.000,E1 309.036} C_DIS
LIN {X 0.037,Y -270.513,Z 1413.703,A 0.000,B 0.000,C 90.000,E1 306.537} C_DIS
LIN {X 0.011,Y -280.002,Z 1413.691,A 0.000,B 0.000,C 90.000,E1 304.452} C_DIS
LIN {X -0.023,Y -286.968,Z 1413.684,A 0.000,B 0.000,C 90.000,E1 303.086} C_DIS
LIN {X 0.020,Y -296.649,Z 1413.674,A 0.000,B 0.000,C 90.000,E1 301.386} C_DIS
LIN {X 0.044,Y -305.264,Z 1413.667,A 0.000,B 0.000,C 90.000,E1 300.050} C_DIS
LIN {X 0.025,Y -314.813,Z 1413.660,A 0.000,B 0.000,C 90.000,E1 298.743} C_DIS
LIN {X 0.012,Y -327.626,Z 1413.651,A 0.000,B 0.000,C 90.000,E1 297.206} C_DIS
LIN {X -0.040,Y -346.787,Z 1413.640,A 0.000,B 0.000,C 90.000,E1 295.155} C_DIS
LIN {X 0.043,Y -359.989,Z 1413.632,A 0.000,B 0.000,C 90.000,E1 293.770} C_DIS
LIN {X 0.095,Y -370.530,Z 1413.626,A 0.000,B 0.000,C 90.000,E1 292.642} C_DIS
LIN {X -0.063,Y -380.826,Z 1413.620,A 0.000,B 0.000,C 90.000,E1 291.535} C_DIS
LIN {X -0.136,Y -393.432,Z 1413.612,A 0.000,B 0.000,C 90.000,E1 290.120} C_DIS
LIN {X -0.218,Y -410.867,Z 1413.601,A 0.000,B 0.000,C 90.000,E1 288.181} C_DIS
LIN {X 0.071,Y -420.774,Z 1413.595,A 0.000,B 0.000,C 90.000,E1 287.040} C_DIS
LIN {X 0.057,Y -425.408,Z 1413.592,A 0.000,B 0.000,C 90.000,E1 286.496} C_DIS
LIN {X -0.049,Y -429.730,Z 1413.589,A 0.000,B 0.000,C 90.000,E1 285.969} C_DIS
LIN {X -0.010,Y -433.630,Z 1413.586,A 0.000,B 0.000,C 90.000,E1 285.426} C_DIS
LIN {X 0.241,Y -438.716,Z 1413.581,A 0.000,B 0.000,C 90.000,E1 284.592} C_DIS
LIN {X 0.009,Y -443.006,Z 1413.577,A 0.000,B 0.000,C 90.000,E1 283.828} C_DIS
LIN {X -0.190,Y -446.539,Z 1413.572,A 0.000,B 0.000,C 90.000,E1 283.063} C_DIS
LIN {X -0.158,Y -448.483,Z 1413.570,A 0.000,B 0.000,C 90.000,E1 282.535} C_DIS
LIN {X -0.119,Y -450.132,Z 1413.567,A 0.000,B 0.000,C 90.000,E1 282.007} C_DIS
LIN {X -0.069,Y -451.426,Z 1413.564,A 0.000,B 0.000,C 90.000,E1 281.478} C_DIS
LIN {X -0.011,Y -452.278,Z 1413.561,A 0.000,B 0.000,C 90.000,E1 280.950} C_DIS
LIN {X -0.029,Y -452.764,Z 1413.558,A 0.000,B 0.000,C 90.000,E1 280.433} C_DIS
LIN {X 0.042,Y -452.731,Z 1413.555,A 0.000,B 0.000,C 90.000,E1 279.905} C_DIS
LIN {X 0.111,Y -452.280,Z 1413.552,A 0.000,B 0.000,C 90.000,E1 279.378} C_DIS
LIN {X 0.106,Y -451.246,Z 1413.549,A 0.000,B 0.000,C 90.000,E1 278.859} C_DIS
LIN {X 0.102,Y -449.644,Z 1413.546,A 0.000,B 0.000,C 90.000,E1 278.341} C_DIS
LIN {X 0.155,Y -447.403,Z 1413.544,A 0.000,B 0.000,C 90.000,E1 277.814} C_DIS
LIN {X 0.130,Y -444.382,Z 1413.541,A 0.000,B 0.000,C 90.000,E1 277.296} C_DIS
LIN {X 0.090,Y -440.495,Z 1413.538,A 0.000,B 0.000,C 90.000,E1 276.777} C_DIS
LIN {X 0.033,Y -435.546,Z 1413.535,A 0.000,B 0.000,C 90.000,E1 276.258} C_DIS
LIN {X 0.064,Y -429.504,Z 1413.532,A 0.000,B 0.000,C 90.000,E1 275.739} C_DIS
LIN {X 0.203,Y -423.176,Z 1413.529,A 0.000,B 0.000,C 90.000,E1 275.277} C_DIS
LIN {X -0.094,Y -416.952,Z 1413.527,A 0.000,B 0.000,C 90.000,E1 274.935} C_DIS
LIN {X -0.088,Y -410.327,Z 1413.525,A 0.000,B 0.000,C 90.000,E1 274.588} C_DIS
LIN {X -0.059,Y -400.212,Z 1413.523,A 0.000,B 0.000,C 90.000,E1 274.131} C_DIS
LIN {X 0.032,Y -390.483,Z 1413.521,A 0.000,B 0.000,C 90.000,E1 273.726} C_DIS
LIN {X -0.053,Y -380.652,Z 1413.519,A 0.000,B 0.000,C 90.000,E1 273.383} C_DIS
LIN {X 0.068,Y -370.440,Z 1413.517,A 0.000,B 0.000,C 90.000,E1 273.037} C_DIS
LIN {X 0.135,Y -360.082,Z 1413.515,A 0.000,B 0.000,C 90.000,E1 272.751} C_DIS
LIN {X 0.124,Y -349.145,Z 1413.514,A 0.000,B 0.000,C 90.000,E1 272.522} C_DIS
LIN {X 0.046,Y -341.339,Z 1413.513,A 0.000,B 0.000,C 90.000,E1 272.407} C_DIS
LIN {X -0.165,Y -326.498,Z 1413.513,A 0.000,B 0.000,C 90.000,E1 272.293} C_DIS
LIN {X 0.148,Y -311.581,Z 1413.512,A 0.000,B 0.000,C 90.000,E1 272.178} C_DIS
LIN {X 0.060,Y -181.230,Z 1413.512,A 0.000,B 0.000,C 90.000,E1 272.178} C_DIS
LIN {X 0.049,Y -181.568,Z 1413.503,A 0.000,B 0.000,C 90.000,E1 270.458} C_DIS
LIN {X -0.091,Y -181.003,Z 1413.484,A 0.000,B 0.000,C 90.000,E1 267.135} C_DIS
LIN {X 0.026,Y -180.907,Z 1413.475,A 0.000,B 0.000,C 90.000,E1 265.412} C_DIS
LIN {X -0.098,Y -180.714,Z 1413.470,A 0.000,B 0.000,C 90.000,E1 264.609} C_DIS
LIN {X 0.001,Y -178.801,Z 1413.442,A 0.000,B 0.000,C 90.000,E1 259.511} C_DIS
LIN {X 0.078,Y -175.846,Z 1413.413,A 0.000,B 0.000,C 90.000,E1 254.393} C_DIS
LIN {X 0.077,Y -172.038,Z 1413.385,A 0.000,B 0.000,C 90.000,E1 249.263} C_DIS
LIN {X 0.053,Y -171.469,Z 1413.380,A 0.000,B 0.000,C 90.000,E1 248.411} C_DIS
LIN {X 0.033,Y -167.701,Z 1413.356,A 0.000,B 0.000,C 90.000,E1 244.101} C_DIS
LIN {X 0.046,Y -166.386,Z 1413.347,A 0.000,B 0.000,C 90.000,E1 242.359} C_DIS
LIN {X 0.038,Y -163.113,Z 1413.327,A 0.000,B 0.000,C 90.000,E1 238.869} C_DIS
LIN {X 0.088,Y -161.062,Z 1413.313,A 0.000,B 0.000,C 90.000,E1 236.215} C_DIS
LIN {X -0.025,Y -157.796,Z 1413.293,A 0.000,B 0.000,C 90.000,E1 232.718} C_DIS
LIN {X 0.014,Y -155.832,Z 1413.278,A 0.000,B 0.000,C 90.000,E1 230.033} C_DIS
LIN {X -0.030,Y -152.082,Z 1413.253,A 0.000,B 0.000,C 90.000,E1 225.567} C_DIS
LIN {X -0.011,Y -150.334,Z 1413.238,A 0.000,B 0.000,C 90.000,E1 222.852} C_DIS
LIN {X 0.010,Y -147.073,Z 1413.213,A 0.000,B 0.000,C 90.000,E1 218.302} C_DIS
LIN {X -0.086,Y -145.647,Z 1413.198,A 0.000,B 0.000,C 90.000,E1 215.598} C_DIS
LIN {X -0.081,Y -143.030,Z 1413.172,A 0.000,B 0.000,C 90.000,E1 211.003} C_DIS
LIN {X 0.046,Y -141.655,Z 1413.151,A 0.000,B 0.000,C 90.000,E1 207.257} C_DIS
LIN {X -0.035,Y -139.445,Z 1413.115,A 0.000,B 0.000,C 90.000,E1 200.791} C_DIS
LIN {X 0.017,Y -139.179,Z 1413.105,A 0.000,B 0.000,C 90.000,E1 198.906} C_DIS
LIN {X 0.046,Y -138.320,Z 1413.053,A 0.000,B 0.000,C 90.000,E1 189.557} C_DIS
LIN {X 0.055,Y -139.467,Z 1413.006,A 0.000,B 0.000,C 90.000,E1 181.146} C_DIS
LIN {X -0.004,Y -141.032,Z 1412.975,A 0.000,B 0.000,C 90.000,E1 175.584} C_DIS
LIN {X -0.050,Y -142.398,Z 1412.960,A 0.000,B 0.000,C 90.000,E1 172.818} C_DIS
LIN {X 0.013,Y -144.631,Z 1412.934,A 0.000,B 0.000,C 90.000,E1 168.173} C_DIS
LIN {X 0.073,Y -147.826,Z 1412.909,A 0.000,B 0.000,C 90.000,E1 163.559} C_DIS
LIN {X 0.017,Y -150.519,Z 1412.889,A 0.000,B 0.000,C 90.000,E1 159.934} C_DIS
LIN {X 0.038,Y -153.981,Z 1412.868,A 0.000,B 0.000,C 90.000,E1 156.305} C_DIS
LIN {X -0.042,Y -157.393,Z 1412.849,A 0.000,B 0.000,C 90.000,E1 152.743} C_DIS
LIN {X 0.039,Y -161.598,Z 1412.829,A 0.000,B 0.000,C 90.000,E1 149.154} C_DIS
LIN {X -0.089,Y -165.795,Z 1412.809,A 0.000,B 0.000,C 90.000,E1 145.674} C_DIS
LIN {X 0.030,Y -170.759,Z 1412.790,A 0.000,B 0.000,C 90.000,E1 142.145} C_DIS
LIN {X 0.053,Y -175.630,Z 1412.771,A 0.000,B 0.000,C 90.000,E1 138.690} C_DIS
LIN {X -0.078,Y -181.245,Z 1412.752,A 0.000,B 0.000,C 90.000,E1 135.324} C_DIS
LIN {X 0.053,Y -186.717,Z 1412.733,A 0.000,B 0.000,C 90.000,E1 131.919} C_DIS
LIN {X 0.004,Y -191.315,Z 1412.719,A 0.000,B 0.000,C 90.000,E1 129.439} C_DIS
LIN {X -0.065,Y -197.146,Z 1412.701,A 0.000,B 0.000,C 90.000,E1 126.171} C_DIS
LIN {X 0.105,Y -199.750,Z 1412.694,A 0.000,B 0.000,C 90.000,E1 124.818} C_DIS
LIN {X 0.110,Y -310.856,Z 1412.694,A 0.000,B 0.000,C 90.000,E1 124.818} C_DIS
LIN {X -0.084,Y -315.802,Z 1412.693,A 0.000,B 0.000,C 90.000,E1 124.692} C_DIS
LIN {X -0.048,Y -318.037,Z 1412.692,A 0.000,B 0.000,C 90.000,E1 124.532} C_DIS
LIN {X -0.024,Y -321.906,Z 1412.690,A 0.000,B 0.000,C 90.000,E1 124.119} C_DIS
LIN {X -0.052,Y -323.811,Z 1412.688,A 0.000,B 0.000,C 90.000,E1 123.833} C_DIS
LIN {X 0.189,Y -325.306,Z 1412.686,A 0.000,B 0.000,C 90.000,E1 123.499} C_DIS
LIN {X 0.105,Y -327.701,Z 1412.683,A 0.000,B 0.000,C 90.000,E1 122.880} C_DIS
LIN {X -0.015,Y -338.314,Z 1412.667,A 0.000,B 0.000,C 90.000,E1 120.079} C_DIS
LIN {X -0.011,Y -350.284,Z 1412.652,A 0.000,B 0.000,C 90.000,E1 117.308} C_DIS
LIN {X 0.011,Y -363.709,Z 1412.637,A 0.000,B 0.000,C 90.000,E1 114.591} C_DIS
LIN {X 0.168,Y -376.961,Z 1412.624,A 0.000,B 0.000,C 90.000,E1 112.206} C_DIS
LIN {X -0.130,Y -391.548,Z 1412.611,A 0.000,B 0.000,C 90.000,E1 109.939} C_DIS
LIN {X 0.174,Y -407.571,Z 1412.598,A 0.000,B 0.000,C 90.000,E1 107.638} C_DIS
LIN {X -0.158,Y -425.144,Z 1412.586,A 0.000,B 0.000,C 90.000,E1 105.481} C_DIS
LIN {X 0.159,Y -444.345,Z 1412.574,A 0.000,B 0.000,C 90.000,E1 103.300} C_DIS
LIN {X 0.204,Y -464.451,Z 1412.563,A 0.000,B 0.000,C 90.000,E1 101.299} C_DIS
LIN {X -0.090,Y -485.043,Z 1412.553,A 0.000,B 0.000,C 90.000,E1 99.500} C_DIS
LIN {X 0.043,Y -487.063,Z 1412.552,A 0.000,B 0.000,C 90.000,E1 99.265} C_DIS
LIN {X -0.065,Y -488.782,Z 1412.550,A 0.000,B 0.000,C 90.000,E1 99.029} C_DIS
LIN {X -0.250,Y -490.068,Z 1412.549,A 0.000,B 0.000,C 90.000,E1 98.803} C_DIS
LIN {X 0.036,Y -491.652,Z 1412.546,A 0.000,B 0.000,C 90.000,E1 98.276} C_DIS
LIN {X 0.257,Y -492.164,Z 1412.543,A 0.000,B 0.000,C 90.000,E1 97.757} C_DIS
LIN {X 0.001,Y -491.688,Z 1412.541,A 0.000,B 0.000,C 90.000,E1 97.296} C_DIS
LIN {X 0.236,Y -490.149,Z 1412.538,A 0.000,B 0.000,C 90.000,E1 96.777} C_DIS
LIN {X 0.081,Y -488.899,Z 1412.536,A 0.000,B 0.000,C 90.000,E1 96.549} C_DIS
LIN {X -0.061,Y -467.863,Z 1412.518,A 0.000,B 0.000,C 90.000,E1 93.326} C_DIS
LIN {X -0.133,Y -459.567,Z 1412.511,A 0.000,B 0.000,C 90.000,E1 92.064} C_DIS
LIN {X 0.183,Y -439.878,Z 1412.494,A 0.000,B 0.000,C 90.000,E1 88.912} C_DIS
LIN {X -0.126,Y -430.690,Z 1412.485,A 0.000,B 0.000,C 90.000,E1 87.364} C_DIS
LIN {X -0.020,Y -419.668,Z 1412.475,A 0.000,B 0.000,C 90.000,E1 85.469} C_DIS
LIN {X -0.116,Y -408.563,Z 1412.464,A 0.000,B 0.000,C 90.000,E1 83.571} C_DIS
LIN {X 0.064,Y -397.405,Z 1412.453,A 0.000,B 0.000,C 90.000,E1 81.602} C_DIS
LIN {X 0.003,Y -386.043,Z 1412.442,A 0.000,B 0.000,C 90.000,E1 79.634} C_DIS
LIN {X -0.151,Y -374.608,Z 1412.431,A 0.000,B 0.000,C 90.000,E1 77.645} C_DIS
LIN {X -0.035,Y -361.667,Z 1412.418,A 0.000,B 0.000,C 90.000,E1 75.283} C_DIS
LIN {X -0.109,Y -351.844,Z 1412.408,A 0.000,B 0.000,C 90.000,E1 73.504} C_DIS
LIN {X 0.169,Y -341.970,Z 1412.398,A 0.000,B 0.000,C 90.000,E1 71.638} C_DIS
LIN {X -0.084,Y -330.322,Z 1412.386,A 0.000,B 0.000,C 90.000,E1 69.518} C_DIS
LIN {X 0.027,Y -317.364,Z 1412.372,A 0.000,B 0.000,C 90.000,E1 66.975} C_DIS
LIN {X -0.052,Y -305.170,Z 1412.358,A 0.000,B 0.000,C 90.000,E1 64.409} C_DIS
LIN {X -0.027,Y -291.580,Z 1412.339,A 0.000,B 0.000,C 90.000,E1 61.101} C_DIS
LIN {X 0.021,Y -279.520,Z 1412.321,A 0.000,B 0.000,C 90.000,E1 57.709} C_DIS
LIN {X -0.017,Y -269.501,Z 1412.303,A 0.000,B 0.000,C 90.000,E1 54.609} C_DIS
LIN {X -0.114,Y -261.165,Z 1412.288,A 0.000,B 0.000,C 90.000,E1 51.823} C_DIS
LIN {X -0.073,Y -251.291,Z 1412.268,A 0.000,B 0.000,C 90.000,E1 48.243} C_DIS
LIN {X -0.042,Y -242.180,Z 1412.248,A 0.000,B 0.000,C 90.000,E1 44.595} C_DIS
LIN {X 0.065,Y -234.008,Z 1412.227,A 0.000,B 0.000,C 90.000,E1 40.862} C_DIS
LIN {X -0.001,Y -226.666,Z 1412.206,A 0.000,B 0.000,C 90.000,E1 37.111} C_DIS
LIN {X -0.025,Y -220.147,Z 1412.185,A 0.000,B 0.000,C 90.000,E1 33.293} C_DIS
LIN {X 0.001,Y -214.523,Z 1412.163,A 0.000,B 0.000,C 90.000,E1 29.411} C_DIS
LIN {X 0.099,Y -209.702,Z 1412.142,A 0.000,B 0.000,C 90.000,E1 25.463} C_DIS
LIN {X -0.009,Y -205.232,Z 1412.115,A 0.000,B 0.000,C 90.000,E1 20.737} C_DIS
LIN {X -0.007,Y -201.454,Z 1412.084,A 0.000,B 0.000,C 90.000,E1 15.134} C_DIS
LIN {X -0.048,Y -199.115,Z 1412.057,A 0.000,B 0.000,C 90.000,E1 10.310} C_DIS
LIN {X -0.034,Y -197.620,Z 1412.035,A 0.000,B 0.000,C 90.000,E1 6.258} C_DIS
LIN {X 0.031,Y -196.477,Z 1412.012,A 0.000,B 0.000,C 90.000,E1 2.178} C_DIS
LIN {X 0.078,Y -195.729,Z 1411.988,A 0.000,B 0.000,C 90.000,E1 357.879} C_DIS
LIN {X 0.091,Y -195.482,Z 1411.966,A 0.000,B 0.000,C 90.000,E1 353.799} C_DIS
LIN {X 0.000,Y -196.007,Z 1411.934,A 0.000,B 0.000,C 90.000,E1 348.117} C_DIS
LIN {X 0.087,Y -198.343,Z 1411.898,A 0.000,B 0.000,C 90.000,E1 341.583} C_DIS
LIN {X 0.042,Y -201.674,Z 1411.871,A 0.000,B 0.000,C 90.000,E1 336.741} C_DIS
LIN {X -0.020,Y -205.719,Z 1411.849,A 0.000,B 0.000,C 90.000,E1 332.743} C_DIS
LIN {X 0.062,Y -210.839,Z 1411.826,A 0.000,B 0.000,C 90.000,E1 328.742} C_DIS
LIN {X 0.050,Y -215.930,Z 1411.809,A 0.000,B 0.000,C 90.000,E1 325.595} C_DIS
LIN {X 0.061,Y -221.997,Z 1411.792,A 0.000,B 0.000,C 90.000,E1 322.477} C_DIS
LIN {X 0.148,Y -228.944,Z 1411.775,A 0.000,B 0.000,C 90.000,E1 319.380} C_DIS
LIN {X -0.163,Y -237.853,Z 1411.756,A 0.000,B 0.000,C 90.000,E1 316.053} C_DIS
LIN {X -0.050,Y -247.953,Z 1411.737,A 0.000,B 0.000,C 90.000,E1 312.690} C_DIS
LIN {X 0.009,Y -257.978,Z 1411.721,A 0.000,B 0.000,C 90.000,E1 309.769} C_DIS
LIN {X -0.133,Y -269.125,Z 1411.705,A 0.000,B 0.000,C 90.000,E1 306.950} C_DIS
LIN {X 0.035,Y -278.441,Z 1411.693,A 0.000,B 0.000,C 90.000,E1 304.818} C_DIS
LIN {X 0.106,Y -287.014,Z 1411.684,A 0.000,B 0.000,C 90.000,E1 303.086} C_DIS
LIN {X -0.001,Y -296.674,Z 1411.675,A 0.000,B 0.000,C 90.000,E1 301.416} C_DIS
LIN {X 0.029,Y -305.283,Z 1411.667,A 0.000,B 0.000,C 90.000,E1 300.079} C_DIS
LIN {X 0.039,Y -314.788,Z 1411.660,A 0.000,B 0.000,C 90.000,E1 298.771} C_DIS
LIN {X -0.175,Y -327.701,Z 1411.651,A 0.000,B 0.000,C 90.000,E1 297.257} C_DIS
LIN {X 0.076,Y -346.808,Z 1411.640,A 0.000,B 0.000,C 90.000,E1 295.155} C_DIS
LIN {X -0.036,Y -360.258,Z 1411.632,A 0.000,B 0.000,C 90.000,E1 293.770} C_DIS
LIN {X 0.050,Y -370.722,Z 1411.626,A 0.000,B 0.000,C 90.000,E1 292.642} C_DIS
LIN {X -0.088,Y -380.991,Z 1411.620,A 0.000,B 0.000,C 90.000,E1 291.535} C_DIS
LIN {X -0.129,Y -393.511,Z 1411.612,A 0.000,B 0.000,C 90.000,E1 290.120} C_DIS
LIN {X 0.102,Y -411.042,Z 1411.601,A 0.000,B 0.000,C 90.000,E1 288.127} C_DIS
LIN {X 0.022,Y -420.926,Z 1411.595,A 0.000,B 0.000,C 90.000,E1 287.040} C_DIS
LIN {X 0.154,Y -427.762,Z 1411.590,A 0.000,B 0.000,C 90.000,E1 286.205} C_DIS
LIN {X -0.057,Y -433.790,Z 1411.586,A 0.000,B 0.000,C 90.000,E1 285.426} C_DIS
LIN {X 0.195,Y -438.920,Z 1411.581,A 0.000,B 0.000,C 90.000,E1 284.592} C_DIS
LIN {X -0.036,Y -443.209,Z 1411.577,A 0.000,B 0.000,C 90.000,E1 283.828} C_DIS
LIN {X -0.234,Y -446.767,Z 1411.572,A 0.000,B 0.000,C 90.000,E1 283.063} C_DIS
LIN {X -0.201,Y -448.677,Z 1411.569,A 0.000,B 0.000,C 90.000,E1 282.535} C_DIS
LIN {X -0.160,Y -450.347,Z 1411.567,A 0.000,B 0.000,C 90.000,E1 282.007} C_DIS
LIN {X -0.110,Y -451.608,Z 1411.564,A 0.000,B 0.000,C 90.000,E1 281.478} C_DIS
LIN {X -0.051,Y -452.526,Z 1411.561,A 0.000,B 0.000,C 90.000,E1 280.950} C_DIS
LIN {X -0.067,Y -453.007,Z 1411.558,A 0.000,B 0.000,C 90.000,E1 280.433} C_DIS
LIN {X 0.004,Y -453.037,Z 1411.555,A 0.000,B 0.000,C 90.000,E1 279.905} C_DIS
LIN {X 0.076,Y -452.548,Z 1411.552,A 0.000,B 0.000,C 90.000,E1 279.378} C_DIS
LIN {X 0.072,Y -451.485,Z 1411.549,A 0.000,B 0.000,C 90.000,E1 278.859} C_DIS
LIN {X 0.070,Y -449.962,Z 1411.546,A 0.000,B 0.000,C 90.000,E1 278.341} C_DIS
LIN {X 0.125,Y -447.742,Z 1411.543,A 0.000,B 0.000,C 90.000,E1 277.814} C_DIS
LIN {X 0.101,Y -444.741,Z 1411.541,A 0.000,B 0.000,C 90.000,E1 277.296} C_DIS
LIN {X 0.064,Y -440.898,Z 1411.538,A 0.000,B 0.000,C 90.000,E1 276.777} C_DIS
LIN {X 0.009,Y -436.037,Z 1411.535,A 0.000,B 0.000,C 90.000,E1 276.258} C_DIS
LIN {X -0.181,Y -433.191,Z 1411.533,A 0.000,B 0.000,C 90.000,E1 276.024} C_DIS
LIN {X 0.063,Y -426.998,Z 1411.531,A 0.000,B 0.000,C 90.000,E1 275.511} C_DIS
LIN {X -0.027,Y -420.694,Z 1411.528,A 0.000,B 0.000,C 90.000,E1 275.106} C_DIS
LIN {X -0.189,Y -414.177,Z 1411.526,A 0.000,B 0.000,C 90.000,E1 274.759} C_DIS
LIN {X -0.072,Y -407.553,Z 1411.525,A 0.000,B 0.000,C 90.000,E1 274.416} C_DIS
LIN {X 0.164,Y -397.680,Z 1411.522,A 0.000,B 0.000,C 90.000,E1 273.955} C_DIS
LIN {X -0.071,Y -387.996,Z 1411.520,A 0.000,B 0.000,C 90.000,E1 273.612} C_DIS
LIN {X -0.109,Y -378.141,Z 1411.518,A 0.000,B 0.000,C 90.000,E1 273.269} C_DIS
LIN {X 0.008,Y -371.287,Z 1411.517,A 0.000,B 0.000,C 90.000,E1 273.037} C_DIS
LIN {X 0.069,Y -360.667,Z 1411.515,A 0.000,B 0.000,C 90.000,E1 272.751} C_DIS
LIN {X 0.051,Y -349.619,Z 1411.514,A 0.000,B 0.000,C 90.000,E1 272.522} C_DIS
LIN {X -0.012,Y -341.843,Z 1411.513,A 0.000,B 0.000,C 90.000,E1 272.407} C_DIS
LIN {X 0.040,Y -332.525,Z 1411.513,A 0.000,B 0.000,C 90.000,E1 272.293} C_DIS
LIN {X -0.005,Y -323.087,Z 1411.512,A 0.000,B 0.000,C 90.000,E1 272.236} C_DIS
LIN {X 0.103,Y -309.395,Z 1411.512,A 0.000,B 0.000,C 90.000,E1 272.178} C_DIS
LIN {X 0.035,Y -181.231,Z 1411.512,A 0.000,B 0.000,C 90.000,E1 272.178} C_DIS
LIN {X 0.024,Y -181.569,Z 1411.503,A 0.000,B 0.000,C 90.000,E1 270.458} C_DIS
LIN {X 0.065,Y -181.002,Z 1411.484,A 0.000,B 0.000,C 90.000,E1 267.078} C_DIS
LIN {X 0.002,Y -180.906,Z 1411.474,A 0.000,B 0.000,C 90.000,E1 265.412} C_DIS
LIN {X 0.058,Y -180.710,Z 1411.470,A 0.000,B 0.000,C 90.000,E1 264.552} C_DIS
LIN {X -0.024,Y -178.797,Z 1411.442,A 0.000,B 0.000,C 90.000,E1 259.511} C_DIS
LIN {X 0.053,Y -175.842,Z 1411.413,A 0.000,B 0.000,C 90.000,E1 254.393} C_DIS
LIN {X 0.053,Y -172.033,Z 1411.385,A 0.000,B 0.000,C 90.000,E1 249.263} C_DIS
LIN {X 0.029,Y -171.463,Z 1411.380,A 0.000,B 0.000,C 90.000,E1 248.411} C_DIS
LIN {X 0.009,Y -167.695,Z 1411.356,A 0.000,B 0.000,C 90.000,E1 244.101} C_DIS
LIN {X 0.023,Y -166.378,Z 1411.346,A 0.000,B 0.000,C 90.000,E1 242.359} C_DIS
LIN {X 0.015,Y -163.106,Z 1411.327,A 0.000,B 0.000,C 90.000,E1 238.869} C_DIS
LIN {X 0.064,Y -161.054,Z 1411.312,A 0.000,B 0.000,C 90.000,E1 236.215} C_DIS
LIN {X 0.048,Y -157.789,Z 1411.293,A 0.000,B 0.000,C 90.000,E1 232.683} C_DIS
LIN {X -0.008,Y -155.826,Z 1411.278,A 0.000,B 0.000,C 90.000,E1 230.033} C_DIS
LIN {X -0.051,Y -152.077,Z 1411.253,A 0.000,B 0.000,C 90.000,E1 225.567} C_DIS
LIN {X -0.032,Y -150.327,Z 1411.238,A 0.000,B 0.000,C 90.000,E1 222.852} C_DIS
LIN {X -0.011,Y -147.068,Z 1411.213,A 0.000,B 0.000,C 90.000,E1 218.302} C_DIS
LIN {X 0.097,Y -145.643,Z 1411.198,A 0.000,B 0.000,C 90.000,E1 215.518} C_DIS
LIN {X 0.094,Y -143.026,Z 1411.172,A 0.000,B 0.000,C 90.000,E1 210.924} C_DIS
LIN {X 0.025,Y -141.652,Z 1411.151,A 0.000,B 0.000,C 90.000,E1 207.257} C_DIS
LIN {X -0.056,Y -139.443,Z 1411.115,A 0.000,B 0.000,C 90.000,E1 200.791} C_DIS
LIN {X -0.003,Y -139.177,Z 1411.105,A 0.000,B 0.000,C 90.000,E1 198.906} C_DIS
LIN {X 0.024,Y -138.320,Z 1411.053,A 0.000,B 0.000,C 90.000,E1 189.557} C_DIS
LIN {X 0.034,Y -139.468,Z 1411.006,A 0.000,B 0.000,C 90.000,E1 181.146} C_DIS
LIN {X -0.025,Y -141.036,Z 1410.975,A 0.000,B 0.000,C 90.000,E1 175.584} C_DIS
LIN {X 0.070,Y -142.403,Z 1410.960,A 0.000,B 0.000,C 90.000,E1 172.761} C_DIS
LIN {X -0.009,Y -144.636,Z 1410.934,A 0.000,B 0.000,C 90.000,E1 168.173} C_DIS
LIN {X 0.051,Y -147.831,Z 1410.909,A 0.000,B 0.000,C 90.000,E1 163.559} C_DIS
LIN {X -0.005,Y -150.526,Z 1410.889,A 0.000,B 0.000,C 90.000,E1 159.934} C_DIS
LIN {X 0.015,Y -153.988,Z 1410.868,A 0.000,B 0.000,C 90.000,E1 156.305} C_DIS
LIN {X -0.064,Y -157.402,Z 1410.848,A 0.000,B 0.000,C 90.000,E1 152.743} C_DIS
LIN {X 0.015,Y -161.609,Z 1410.829,A 0.000,B 0.000,C 90.000,E1 149.154} C_DIS
LIN {X -0.019,Y -165.805,Z 1410.809,A 0.000,B 0.000,C 90.000,E1 145.642} C_DIS
LIN {X 0.006,Y -170.771,Z 1410.790,A 0.000,B 0.000,C 90.000,E1 142.145} C_DIS
LIN {X 0.029,Y -175.642,Z 1410.771,A 0.000,B 0.000,C 90.000,E1 138.690} C_DIS
LIN {X -0.103,Y -181.257,Z 1410.752,A 0.000,B 0.000,C 90.000,E1 135.324} C_DIS
LIN {X 0.028,Y -186.730,Z 1410.733,A 0.000,B 0.000,C 90.000,E1 131.919} C_DIS
LIN {X -0.022,Y -191.327,Z 1410.719,A 0.000,B 0.000,C 90.000,E1 129.439} C_DIS
LIN {X 0.025,Y -197.160,Z 1410.701,A 0.000,B 0.000,C 90.000,E1 126.137} C_DIS
LIN {X -0.090,Y -199.701,Z 1410.694,A 0.000,B 0.000,C 90.000,E1 124.898} C_DIS
LIN {X -0.022,Y -310.361,Z 1410.694,A 0.000,B 0.000,C 90.000,E1 124.865} C_DIS
LIN {X -0.015,Y -315.834,Z 1410.693,A 0.000,B 0.000,C 90.000,E1 124.692} C_DIS
LIN {X -0.089,Y -318.274,Z 1410.692,A 0.000,B 0.000,C 90.000,E1 124.532} C_DIS
LIN {X -0.136,Y -322.105,Z 1410.689,A 0.000,B 0.000,C 90.000,E1 124.119} C_DIS
LIN {X 0.055,Y -323.993,Z 1410.688,A 0.000,B 0.000,C 90.000,E1 123.785} C_DIS
LIN {X -0.024,Y -325.473,Z 1410.686,A 0.000,B 0.000,C 90.000,E1 123.499} C_DIS
LIN {X 0.049,Y -332.374,Z 1410.676,A 0.000,B 0.000,C 90.000,E1 121.592} C_DIS
LIN {X -0.111,Y -343.595,Z 1410.660,A 0.000,B 0.000,C 90.000,E1 118.821} C_DIS
LIN {X 0.029,Y -356.218,Z 1410.645,A 0.000,B 0.000,C 90.000,E1 116.052} C_DIS
LIN {X -0.103,Y -370.347,Z 1410.630,A 0.000,B 0.000,C 90.000,E1 113.387} C_DIS
LIN {X -0.074,Y -384.274,Z 1410.617,A 0.000,B 0.000,C 90.000,E1 111.046} C_DIS
LIN {X 0.181,Y -399.587,Z 1410.604,A 0.000,B 0.000,C 90.000,E1 108.725} C_DIS
LIN {X 0.181,Y -416.392,Z 1410.592,A 0.000,B 0.000,C 90.000,E1 106.496} C_DIS
LIN {X -0.057,Y -434.809,Z 1410.580,A 0.000,B 0.000,C 90.000,E1 104.356} C_DIS
LIN {X -0.221,Y -454.598,Z 1410.568,A 0.000,B 0.000,C 90.000,E1 102.299} C_DIS
LIN {X -0.053,Y -474.990,Z 1410.557,A 0.000,B 0.000,C 90.000,E1 100.366} C_DIS
LIN {X 0.166,Y -485.272,Z 1410.553,A 0.000,B 0.000,C 90.000,E1 99.443} C_DIS
LIN {X -0.179,Y -487.199,Z 1410.551,A 0.000,B 0.000,C 90.000,E1 99.265} C_DIS
LIN {X 0.195,Y -488.848,Z 1410.550,A 0.000,B 0.000,C 90.000,E1 98.973} C_DIS
LIN {X 0.012,Y -490.081,Z 1410.549,A 0.000,B 0.000,C 90.000,E1 98.746} C_DIS
LIN {X -0.187,Y -491.581,Z 1410.546,A 0.000,B 0.000,C 90.000,E1 98.276} C_DIS
LIN {X 0.035,Y -492.021,Z 1410.543,A 0.000,B 0.000,C 90.000,E1 97.757} C_DIS
LIN {X -0.221,Y -491.475,Z 1410.540,A 0.000,B 0.000,C 90.000,E1 97.296} C_DIS
LIN {X 0.014,Y -489.854,Z 1410.538,A 0.000,B 0.000,C 90.000,E1 96.777} C_DIS
LIN {X -0.087,Y -488.551,Z 1410.536,A 0.000,B 0.000,C 90.000,E1 96.543} C_DIS
LIN {X -0.095,Y -469.063,Z 1410.520,A 0.000,B 0.000,C 90.000,E1 93.555} C_DIS
LIN {X -0.147,Y -460.854,Z 1410.513,A 0.000,B 0.000,C 90.000,E1 92.293} C_DIS
LIN {X -0.049,Y -439.514,Z 1410.494,A 0.000,B 0.000,C 90.000,E1 88.912} C_DIS
LIN {X 0.071,Y -430.349,Z 1410.485,A 0.000,B 0.000,C 90.000,E1 87.306} C_DIS
LIN {X 0.164,Y -419.379,Z 1410.475,A 0.000,B 0.000,C 90.000,E1 85.412} C_DIS
LIN {X 0.056,Y -408.286,Z 1410.464,A 0.000,B 0.000,C 90.000,E1 83.514} C_DIS
LIN {X 0.140,Y -398.749,Z 1410.455,A 0.000,B 0.000,C 90.000,E1 81.837} C_DIS
LIN {X 0.117,Y -389.057,Z 1410.445,A 0.000,B 0.000,C 90.000,E1 80.151} C_DIS
LIN {X -0.048,Y -377.656,Z 1410.434,A 0.000,B 0.000,C 90.000,E1 78.173} C_DIS
LIN {X 0.048,Y -364.658,Z 1410.421,A 0.000,B 0.000,C 90.000,E1 75.825} C_DIS
LIN {X 0.021,Y -354.896,Z 1410.411,A 0.000,B 0.000,C 90.000,E1 74.047} C_DIS
LIN {X 0.020,Y -345.012,Z 1410.401,A 0.000,B 0.000,C 90.000,E1 72.236} C_DIS
LIN {X -0.148,Y -335.055,Z 1410.391,A 0.000,B 0.000,C 90.000,E1 70.423} C_DIS
LIN {X -0.083,Y -320.299,Z 1410.375,A 0.000,B 0.000,C 90.000,E1 67.592} C_DIS
LIN {X 0.108,Y -306.390,Z 1410.359,A 0.000,B 0.000,C 90.000,E1 64.665} C_DIS
LIN {X 0.017,Y -293.966,Z 1410.343,A 0.000,B 0.000,C 90.000,E1 61.719} C_DIS
LIN {X 0.122,Y -281.662,Z 1410.324,A 0.000,B 0.000,C 90.000,E1 58.329} C_DIS
LIN {X -0.019,Y -271.544,Z 1410.307,A 0.000,B 0.000,C 90.000,E1 55.261} C_DIS
LIN {X 0.050,Y -261.085,Z 1410.287,A 0.000,B 0.000,C 90.000,E1 51.743} C_DIS
LIN {X 0.085,Y -251.242,Z 1410.268,A 0.000,B 0.000,C 90.000,E1 48.162} C_DIS
LIN {X 0.111,Y -242.165,Z 1410.247,A 0.000,B 0.000,C 90.000,E1 44.514} C_DIS
LIN {X 0.033,Y -234.016,Z 1410.227,A 0.000,B 0.000,C 90.000,E1 40.825} C_DIS
LIN {X -0.042,Y -226.708,Z 1410.206,A 0.000,B 0.000,C 90.000,E1 37.076} C_DIS
LIN {X -0.013,Y -220.219,Z 1410.185,A 0.000,B 0.000,C 90.000,E1 33.245} C_DIS
LIN {X 0.022,Y -214.632,Z 1410.163,A 0.000,B 0.000,C 90.000,E1 29.361} C_DIS
LIN {X -0.059,Y -209.859,Z 1410.141,A 0.000,B 0.000,C 90.000,E1 25.463} C_DIS
LIN {X 0.034,Y -205.452,Z 1410.115,A 0.000,B 0.000,C 90.000,E1 20.684} C_DIS
LIN {X -0.006,Y -202.200,Z 1410.088,A 0.000,B 0.000,C 90.000,E1 15.898} C_DIS
LIN {X -0.020,Y -199.750,Z 1410.062,A 0.000,B 0.000,C 90.000,E1 11.074} C_DIS
LIN {X 0.049,Y -198.216,Z 1410.039,A 0.000,B 0.000,C 90.000,E1 7.011} C_DIS
LIN {X -0.073,Y -196.787,Z 1410.012,A 0.000,B 0.000,C 90.000,E1 2.178} C_DIS
LIN {X 0.038,Y -195.942,Z 1409.984,A 0.000,B 0.000,C 90.000,E1 357.078} C_DIS
LIN {X 0.045,Y -195.773,Z 1409.957,A 0.000,B 0.000,C 90.000,E1 352.186} C_DIS
LIN {X 0.108,Y -196.620,Z 1409.925,A 0.000,B 0.000,C 90.000,E1 346.464} C_DIS
LIN {X -0.032,Y -199.499,Z 1409.889,A 0.000,B 0.000,C 90.000,E1 340.007} C_DIS
LIN {X 0.015,Y -203.390,Z 1409.862,A 0.000,B 0.000,C 90.000,E1 335.153} C_DIS
LIN {X -0.081,Y -207.863,Z 1409.840,A 0.000,B 0.000,C 90.000,E1 331.179} C_DIS
LIN {X -0.008,Y -213.492,Z 1409.818,A 0.000,B 0.000,C 90.000,E1 327.199} C_DIS
LIN {X -0.017,Y -219.048,Z 1409.800,A 0.000,B 0.000,C 90.000,E1 324.069} C_DIS
LIN {X 0.023,Y -225.547,Z 1409.783,A 0.000,B 0.000,C 90.000,E1 320.964} C_DIS
LIN {X -0.052,Y -233.926,Z 1409.764,A 0.000,B 0.000,C 90.000,E1 317.553} C_DIS
LIN {X -0.059,Y -243.456,Z 1409.745,A 0.000,B 0.000,C 90.000,E1 314.190} C_DIS
LIN {X 0.074,Y -254.211,Z 1409.727,A 0.000,B 0.000,C 90.000,E1 310.862} C_DIS
LIN {X 0.020,Y -266.308,Z 1409.709,A 0.000,B 0.000,C 90.000,E1 307.649} C_DIS
LIN {X 0.066,Y -276.903,Z 1409.696,A 0.000,B 0.000,C 90.000,E1 305.185} C_DIS
LIN {X -0.126,Y -285.278,Z 1409.686,A 0.000,B 0.000,C 90.000,E1 303.499} C_DIS
LIN {X -0.107,Y -294.684,Z 1409.677,A 0.000,B 0.000,C 90.000,E1 301.799} C_DIS
LIN {X -0.110,Y -303.069,Z 1409.669,A 0.000,B 0.000,C 90.000,E1 300.463} C_DIS
LIN {X -0.006,Y -312.321,Z 1409.662,A 0.000,B 0.000,C 90.000,E1 299.127} C_DIS
LIN {X 0.064,Y -325.345,Z 1409.653,A 0.000,B 0.000,C 90.000,E1 297.513} C_DIS
LIN {X 0.069,Y -347.032,Z 1409.640,A 0.000,B 0.000,C 90.000,E1 295.155} C_DIS
LIN {X -0.108,Y -360.515,Z 1409.632,A 0.000,B 0.000,C 90.000,E1 293.770} C_DIS
LIN {X -0.078,Y -371.039,Z 1409.626,A 0.000,B 0.000,C 90.000,E1 292.642} C_DIS
LIN {X 0.089,Y -381.362,Z 1409.619,A 0.000,B 0.000,C 90.000,E1 291.482} C_DIS
LIN {X -0.027,Y -393.951,Z 1409.611,A 0.000,B 0.000,C 90.000,E1 290.066} C_DIS
LIN {X -0.075,Y -411.511,Z 1409.601,A 0.000,B 0.000,C 90.000,E1 288.109} C_DIS
LIN {X -0.213,Y -421.305,Z 1409.594,A 0.000,B 0.000,C 90.000,E1 287.040} C_DIS
LIN {X -0.081,Y -428.145,Z 1409.590,A 0.000,B 0.000,C 90.000,E1 286.205} C_DIS
LIN {X -0.052,Y -432.236,Z 1409.587,A 0.000,B 0.000,C 90.000,E1 285.662} C_DIS
LIN {X 0.191,Y -437.650,Z 1409.583,A 0.000,B 0.000,C 90.000,E1 284.828} C_DIS
LIN {X -0.057,Y -442.204,Z 1409.578,A 0.000,B 0.000,C 90.000,E1 284.064} C_DIS
LIN {X 0.175,Y -445.981,Z 1409.574,A 0.000,B 0.000,C 90.000,E1 283.244} C_DIS
LIN {X 0.005,Y -448.993,Z 1409.569,A 0.000,B 0.000,C 90.000,E1 282.479} C_DIS
LIN {X 0.048,Y -450.611,Z 1409.566,A 0.000,B 0.000,C 90.000,E1 281.951} C_DIS
LIN {X 0.103,Y -451.880,Z 1409.563,A 0.000,B 0.000,C 90.000,E1 281.422} C_DIS
LIN {X 0.165,Y -452.794,Z 1409.561,A 0.000,B 0.000,C 90.000,E1 280.894} C_DIS
LIN {X 0.232,Y -453.234,Z 1409.558,A 0.000,B 0.000,C 90.000,E1 280.366} C_DIS
LIN {X -0.221,Y -453.236,Z 1409.555,A 0.000,B 0.000,C 90.000,E1 279.905} C_DIS
LIN {X -0.149,Y -452.758,Z 1409.552,A 0.000,B 0.000,C 90.000,E1 279.378} C_DIS
LIN {X -0.151,Y -451.709,Z 1409.549,A 0.000,B 0.000,C 90.000,E1 278.859} C_DIS
LIN {X -0.151,Y -450.178,Z 1409.546,A 0.000,B 0.000,C 90.000,E1 278.341} C_DIS
LIN {X -0.094,Y -447.945,Z 1409.543,A 0.000,B 0.000,C 90.000,E1 277.814} C_DIS
LIN {X -0.115,Y -444.943,Z 1409.540,A 0.000,B 0.000,C 90.000,E1 277.296} C_DIS
LIN {X 0.115,Y -443.141,Z 1409.539,A 0.000,B 0.000,C 90.000,E1 277.004} C_DIS
LIN {X 0.068,Y -438.819,Z 1409.536,A 0.000,B 0.000,C 90.000,E1 276.486} C_DIS
LIN {X -0.201,Y -436.253,Z 1409.535,A 0.000,B 0.000,C 90.000,E1 276.258} C_DIS
LIN {X -0.178,Y -430.254,Z 1409.532,A 0.000,B 0.000,C 90.000,E1 275.739} C_DIS
LIN {X -0.078,Y -423.984,Z 1409.529,A 0.000,B 0.000,C 90.000,E1 275.277} C_DIS
LIN {X -0.016,Y -417.557,Z 1409.527,A 0.000,B 0.000,C 90.000,E1 274.878} C_DIS
LIN {X -0.019,Y -410.945,Z 1409.525,A 0.000,B 0.000,C 90.000,E1 274.531} C_DIS
LIN {X 0.092,Y -401.196,Z 1409.523,A 0.000,B 0.000,C 90.000,E1 274.073} C_DIS
LIN {X 0.151,Y -391.386,Z 1409.521,A 0.000,B 0.000,C 90.000,E1 273.669} C_DIS
LIN {X 0.092,Y -381.764,Z 1409.519,A 0.000,B 0.000,C 90.000,E1 273.326} C_DIS
LIN {X -0.133,Y -371.640,Z 1409.517,A 0.000,B 0.000,C 90.000,E1 273.037} C_DIS
LIN {X -0.069,Y -360.905,Z 1409.515,A 0.000,B 0.000,C 90.000,E1 272.751} C_DIS
LIN {X 0.035,Y -353.808,Z 1409.514,A 0.000,B 0.000,C 90.000,E1 272.579} C_DIS
LIN {X -0.096,Y -342.154,Z 1409.513,A 0.000,B 0.000,C 90.000,E1 272.407} C_DIS
LIN {X -0.041,Y -332.625,Z 1409.513,A 0.000,B 0.000,C 90.000,E1 272.293} C_DIS
LIN {X -0.143,Y -318.392,Z 1409.512,A 0.000,B 0.000,C 90.000,E1 272.236} C_DIS
LIN {X 0.075,Y -309.229,Z 1409.512,A 0.000,B 0.000,C 90.000,E1 272.178} C_DIS
LIN {X 0.023,Y -181.233,Z 1409.512,A 0.000,B 0.000,C 90.000,E1 272.178} C_DIS
LIN {X 0.009,Y -181.570,Z 1409.503,A 0.000,B 0.000,C 90.000,E1 270.458} C_DIS
LIN {X 0.050,Y -181.002,Z 1409.484,A 0.000,B 0.000,C 90.000,E1 267.078} C_DIS
LIN {X -0.013,Y -180.907,Z 1409.474,A 0.000,B 0.000,C 90.000,E1 265.412} C_DIS
LIN {X 0.044,Y -180.708,Z 1409.470,A 0.000,B 0.000,C 90.000,E1 264.552} C_DIS
LIN {X -0.038,Y -178.794,Z 1409.442,A 0.000,B 0.000,C 90.000,E1 259.511} C_DIS
LIN {X 0.039,Y -175.840,Z 1409.413,A 0.000,B 0.000,C 90.000,E1 254.393} C_DIS
LIN {X 0.039,Y -172.030,Z 1409.385,A 0.000,B 0.000,C 90.000,E1 249.263} C_DIS
LIN {X 0.015,Y -171.458,Z 1409.380,A 0.000,B 0.000,C 90.000,E1 248.411} C_DIS
LIN {X -0.005,Y -167.691,Z 1409.356,A 0.000,B 0.000,C 90.000,E1 244.101} C_DIS
LIN {X 0.009,Y -166.373,Z 1409.346,A 0.000,B 0.000,C 90.000,E1 242.359} C_DIS
LIN {X 0.001,Y -163.103,Z 1409.327,A 0.000,B 0.000,C 90.000,E1 238.869} C_DIS
LIN {X 0.052,Y -161.049,Z 1409.312,A 0.000,B 0.000,C 90.000,E1 236.215} C_DIS
LIN {X 0.035,Y -157.786,Z 1409.293,A 0.000,B 0.000,C 90.000,E1 232.683} C_DIS
LIN {X -0.022,Y -155.822,Z 1409.278,A 0.000,B 0.000,C 90.000,E1 230.033} C_DIS
LIN {X -0.065,Y -152.073,Z 1409.253,A 0.000,B 0.000,C 90.000,E1 225.567} C_DIS
LIN {X -0.045,Y -150.324,Z 1409.238,A 0.000,B 0.000,C 90.000,E1 222.852} C_DIS
LIN {X -0.024,Y -147.065,Z 1409.213,A 0.000,B 0.000,C 90.000,E1 218.302} C_DIS
LIN {X 0.084,Y -145.641,Z 1409.198,A 0.000,B 0.000,C 90.000,E1 215.518} C_DIS
LIN {X 0.082,Y -143.023,Z 1409.172,A 0.000,B 0.000,C 90.000,E1 210.924} C_DIS
LIN {X 0.012,Y -141.649,Z 1409.151,A 0.000,B 0.000,C 90.000,E1 207.257} C_DIS
LIN {X 0.062,Y -139.443,Z 1409.115,A 0.000,B 0.000,C 90.000,E1 200.737} C_DIS
LIN {X -0.015,Y -139.176,Z 1409.105,A 0.000,B 0.000,C 90.000,E1 198.906} C_DIS
LIN {X 0.012,Y -138.319,Z 1409.053,A 0.000,B 0.000,C 90.000,E1 189.557} C_DIS
LIN {X 0.022,Y -139.468,Z 1409.006,A 0.000,B 0.000,C 90.000,E1 181.146} C_DIS
LIN {X -0.038,Y -141.038,Z 1408.975,A 0.000,B 0.000,C 90.000,E1 175.584} C_DIS
LIN {X 0.057,Y -142.406,Z 1408.960,A 0.000,B 0.000,C 90.000,E1 172.761} C_DIS
LIN {X -0.021,Y -144.639,Z 1408.934,A 0.000,B 0.000,C 90.000,E1 168.173} C_DIS
LIN {X 0.038,Y -147.834,Z 1408.909,A 0.000,B 0.000,C 90.000,E1 163.559} C_DIS
LIN {X -0.017,Y -150.530,Z 1408.888,A 0.000,B 0.000,C 90.000,E1 159.934} C_DIS
LIN {X 0.002,Y -153.993,Z 1408.868,A 0.000,B 0.000,C 90.000,E1 156.305} C_DIS
LIN {X -0.078,Y -157.407,Z 1408.848,A 0.000,B 0.000,C 90.000,E1 152.743} C_DIS
LIN {X 0.002,Y -161.616,Z 1408.829,A 0.000,B 0.000,C 90.000,E1 149.154} C_DIS
LIN {X 0.103,Y -165.811,Z 1408.809,A 0.000,B 0.000,C 90.000,E1 145.595} C_DIS
LIN {X -0.008,Y -170.778,Z 1408.790,A 0.000,B 0.000,C 90.000,E1 142.145} C_DIS
LIN {X 0.015,Y -175.650,Z 1408.771,A 0.000,B 0.000,C 90.000,E1 138.690} C_DIS
LIN {X 0.012,Y -181.264,Z 1408.752,A 0.000,B 0.000,C 90.000,E1 135.283} C_DIS
LIN {X 0.013,Y -186.738,Z 1408.733,A 0.000,B 0.000,C 90.000,E1 131.919} C_DIS
LIN {X -0.037,Y -191.334,Z 1408.719,A 0.000,B 0.000,C 90.000,E1 129.439} C_DIS
LIN {X 0.010,Y -197.169,Z 1408.701,A 0.000,B 0.000,C 90.000,E1 126.137} C_DIS
LIN {X -0.027,Y -199.663,Z 1408.694,A 0.000,B 0.000,C 90.000,E1 124.898} C_DIS
LIN {X -0.102,Y -310.543,Z 1408.694,A 0.000,B 0.000,C 90.000,E1 124.898} C_DIS
LIN {X -0.044,Y -311.983,Z 1408.694,A 0.000,B 0.000,C 90.000,E1 124.865} C_DIS
LIN {X -0.038,Y -316.144,Z 1408.693,A 0.000,B 0.000,C 90.000,E1 124.692} C_DIS
LIN {X -0.113,Y -318.462,Z 1408.692,A 0.000,B 0.000,C 90.000,E1 124.532} C_DIS
LIN {X -0.004,Y -322.320,Z 1408.689,A 0.000,B 0.000,C 90.000,E1 124.072} C_DIS
LIN {X -0.127,Y -324.184,Z 1408.688,A 0.000,B 0.000,C 90.000,E1 123.785} C_DIS
LIN {X 0.020,Y -325.641,Z 1408.686,A 0.000,B 0.000,C 90.000,E1 123.452} C_DIS
LIN {X -0.002,Y -338.578,Z 1408.667,A 0.000,B 0.000,C 90.000,E1 120.001} C_DIS
LIN {X -0.157,Y -350.586,Z 1408.651,A 0.000,B 0.000,C 90.000,E1 117.257} C_DIS
LIN {X 0.027,Y -364.051,Z 1408.636,A 0.000,B 0.000,C 90.000,E1 114.515} C_DIS
LIN {X 0.043,Y -377.343,Z 1408.623,A 0.000,B 0.000,C 90.000,E1 112.153} C_DIS
LIN {X -0.111,Y -391.971,Z 1408.610,A 0.000,B 0.000,C 90.000,E1 109.866} C_DIS
LIN {X 0.071,Y -408.040,Z 1408.598,A 0.000,B 0.000,C 90.000,E1 107.583} C_DIS
LIN {X 0.162,Y -425.661,Z 1408.586,A 0.000,B 0.000,C 90.000,E1 105.371} C_DIS
LIN {X 0.092,Y -444.903,Z 1408.574,A 0.000,B 0.000,C 90.000,E1 103.244} C_DIS
LIN {X 0.177,Y -465.028,Z 1408.563,A 0.000,B 0.000,C 90.000,E1 101.243} C_DIS
LIN {X -0.075,Y -485.500,Z 1408.552,A 0.000,B 0.000,C 90.000,E1 99.443} C_DIS
LIN {X 0.062,Y -487.336,Z 1408.551,A 0.000,B 0.000,C 90.000,E1 99.208} C_DIS
LIN {X -0.045,Y -488.913,Z 1408.550,A 0.000,B 0.000,C 90.000,E1 98.973} C_DIS
LIN {X -0.227,Y -490.090,Z 1408.548,A 0.000,B 0.000,C 90.000,E1 98.746} C_DIS
LIN {X 0.059,Y -491.505,Z 1408.546,A 0.000,B 0.000,C 90.000,E1 98.219} C_DIS
LIN {X -0.206,Y -491.871,Z 1408.543,A 0.000,B 0.000,C 90.000,E1 97.757} C_DIS
LIN {X 0.025,Y -491.249,Z 1408.540,A 0.000,B 0.000,C 90.000,E1 97.239} C_DIS
LIN {X -0.227,Y -489.538,Z 1408.537,A 0.000,B 0.000,C 90.000,E1 96.777} C_DIS
LIN {X 0.158,Y -488.176,Z 1408.536,A 0.000,B 0.000,C 90.000,E1 96.486} C_DIS
LIN {X 0.129,Y -468.638,Z 1408.520,A 0.000,B 0.000,C 90.000,E1 93.498} C_DIS
LIN {X -0.185,Y -462.115,Z 1408.514,A 0.000,B 0.000,C 90.000,E1 92.522} C_DIS
LIN {X 0.218,Y -442.245,Z 1408.497,A 0.000,B 0.000,C 90.000,E1 89.370} C_DIS
LIN {X -0.179,Y -429.989,Z 1408.485,A 0.000,B 0.000,C 90.000,E1 87.306} C_DIS
LIN {X -0.087,Y -419.070,Z 1408.474,A 0.000,B 0.000,C 90.000,E1 85.412} C_DIS
LIN {X -0.193,Y -408.003,Z 1408.464,A 0.000,B 0.000,C 90.000,E1 83.514} C_DIS
LIN {X -0.109,Y -398.491,Z 1408.455,A 0.000,B 0.000,C 90.000,E1 81.837} C_DIS
LIN {X -0.131,Y -388.814,Z 1408.445,A 0.000,B 0.000,C 90.000,E1 80.151} C_DIS
LIN {X 0.076,Y -377.445,Z 1408.434,A 0.000,B 0.000,C 90.000,E1 78.117} C_DIS
LIN {X -0.104,Y -364.447,Z 1408.421,A 0.000,B 0.000,C 90.000,E1 75.811} C_DIS
LIN {X -0.121,Y -354.628,Z 1408.411,A 0.000,B 0.000,C 90.000,E1 74.031} C_DIS
LIN {X 0.111,Y -344.740,Z 1408.401,A 0.000,B 0.000,C 90.000,E1 72.181} C_DIS
LIN {X -0.068,Y -334.776,Z 1408.391,A 0.000,B 0.000,C 90.000,E1 70.369} C_DIS
LIN {X -0.070,Y -318.433,Z 1408.373,A 0.000,B 0.000,C 90.000,E1 67.230} C_DIS
LIN {X -0.088,Y -304.687,Z 1408.357,A 0.000,B 0.000,C 90.000,E1 64.332} C_DIS
LIN {X 0.050,Y -292.445,Z 1408.341,A 0.000,B 0.000,C 90.000,E1 61.335} C_DIS
LIN {X -0.135,Y -280.315,Z 1408.322,A 0.000,B 0.000,C 90.000,E1 57.995} C_DIS
LIN {X 0.139,Y -271.410,Z 1408.307,A 0.000,B 0.000,C 90.000,E1 55.182} C_DIS
LIN {X 0.039,Y -261.002,Z 1408.287,A 0.000,B 0.000,C 90.000,E1 51.698} C_DIS
LIN {X -0.125,Y -251.188,Z 1408.267,A 0.000,B 0.000,C 90.000,E1 48.162} C_DIS
LIN {X -0.094,Y -242.141,Z 1408.247,A 0.000,B 0.000,C 90.000,E1 44.514} C_DIS
LIN {X 0.012,Y -234.018,Z 1408.227,A 0.000,B 0.000,C 90.000,E1 40.782} C_DIS
LIN {X -0.053,Y -226.748,Z 1408.206,A 0.000,B 0.000,C 90.000,E1 37.030} C_DIS
LIN {X 0.108,Y -220.291,Z 1408.184,A 0.000,B 0.000,C 90.000,E1 33.166} C_DIS
LIN {X -0.050,Y -214.726,Z 1408.163,A 0.000,B 0.000,C 90.000,E1 29.333} C_DIS
LIN {X -0.040,Y -210.020,Z 1408.141,A 0.000,B 0.000,C 90.000,E1 25.412} C_DIS
LIN {X -0.053,Y -205.672,Z 1408.115,A 0.000,B 0.000,C 90.000,E1 20.663} C_DIS
LIN {X 0.039,Y -202.468,Z 1408.088,A 0.000,B 0.000,C 90.000,E1 15.843} C_DIS
LIN {X 0.029,Y -200.428,Z 1408.066,A 0.000,B 0.000,C 90.000,E1 11.827} C_DIS
LIN {X -0.056,Y -198.820,Z 1408.043,A 0.000,B 0.000,C 90.000,E1 7.814} C_DIS
LIN {X 0.073,Y -197.483,Z 1408.021,A 0.000,B 0.000,C 90.000,E1 3.726} C_DIS
LIN {X -0.035,Y -196.575,Z 1407.997,A 0.000,B 0.000,C 90.000,E1 359.542} C_DIS
LIN {X -0.026,Y -196.079,Z 1407.975,A 0.000,B 0.000,C 90.000,E1 355.469} C_DIS
LIN {X 0.046,Y -196.255,Z 1407.943,A 0.000,B 0.000,C 90.000,E1 349.746} C_DIS
LIN {X 0.081,Y -198.407,Z 1407.902,A 0.000,B 0.000,C 90.000,E1 342.417} C_DIS
LIN {X -0.022,Y -201.468,Z 1407.875,A 0.000,B 0.000,C 90.000,E1 337.592} C_DIS
LIN {X 0.016,Y -205.283,Z 1407.853,A 0.000,B 0.000,C 90.000,E1 333.563} C_DIS
LIN {X -0.008,Y -210.170,Z 1407.831,A 0.000,B 0.000,C 90.000,E1 329.587} C_DIS
LIN {X -0.109,Y -216.357,Z 1407.809,A 0.000,B 0.000,C 90.000,E1 325.674} C_DIS
LIN {X -0.095,Y -222.391,Z 1407.792,A 0.000,B 0.000,C 90.000,E1 322.557} C_DIS
LIN {X -0.004,Y -229.324,Z 1407.775,A 0.000,B 0.000,C 90.000,E1 319.461} C_DIS
LIN {X 0.025,Y -238.170,Z 1407.756,A 0.000,B 0.000,C 90.000,E1 316.053} C_DIS
LIN {X 0.154,Y -248.189,Z 1407.737,A 0.000,B 0.000,C 90.000,E1 312.690} C_DIS
LIN {X 0.064,Y -258.235,Z 1407.721,A 0.000,B 0.000,C 90.000,E1 309.806} C_DIS
LIN {X 0.102,Y -269.325,Z 1407.705,A 0.000,B 0.000,C 90.000,E1 306.950} C_DIS
LIN {X -0.107,Y -278.577,Z 1407.694,A 0.000,B 0.000,C 90.000,E1 304.898} C_DIS
LIN {X -0.035,Y -287.120,Z 1407.684,A 0.000,B 0.000,C 90.000,E1 303.166} C_DIS
LIN {X 0.013,Y -296.709,Z 1407.675,A 0.000,B 0.000,C 90.000,E1 301.465} C_DIS
LIN {X 0.040,Y -305.324,Z 1407.667,A 0.000,B 0.000,C 90.000,E1 300.129} C_DIS
LIN {X 0.025,Y -314.837,Z 1407.660,A 0.000,B 0.000,C 90.000,E1 298.821} C_DIS
LIN {X -0.127,Y -328.116,Z 1407.651,A 0.000,B 0.000,C 90.000,E1 297.257} C_DIS
LIN {X 0.024,Y -347.295,Z 1407.640,A 0.000,B 0.000,C 90.000,E1 295.155} C_DIS
LIN {X -0.196,Y -360.806,Z 1407.632,A 0.000,B 0.000,C 90.000,E1 293.770} C_DIS
LIN {X -0.187,Y -371.330,Z 1407.626,A 0.000,B 0.000,C 90.000,E1 292.642} C_DIS
LIN {X 0.081,Y -381.664,Z 1407.619,A 0.000,B 0.000,C 90.000,E1 291.461} C_DIS
LIN {X -0.196,Y -394.264,Z 1407.611,A 0.000,B 0.000,C 90.000,E1 290.066} C_DIS
LIN {X 0.157,Y -411.785,Z 1407.600,A 0.000,B 0.000,C 90.000,E1 288.055} C_DIS
LIN {X -0.026,Y -421.646,Z 1407.594,A 0.000,B 0.000,C 90.000,E1 286.985} C_DIS
LIN {X 0.114,Y -428.458,Z 1407.590,A 0.000,B 0.000,C 90.000,E1 286.150} C_DIS
LIN {X 0.147,Y -432.549,Z 1407.587,A 0.000,B 0.000,C 90.000,E1 285.607} C_DIS
LIN {X -0.027,Y -437.972,Z 1407.582,A 0.000,B 0.000,C 90.000,E1 284.828} C_DIS
LIN {X 0.156,Y -442.539,Z 1407.578,A 0.000,B 0.000,C 90.000,E1 284.008} C_DIS
LIN {X -0.041,Y -446.288,Z 1407.574,A 0.000,B 0.000,C 90.000,E1 283.244} C_DIS
LIN {X -0.209,Y -449.287,Z 1407.569,A 0.000,B 0.000,C 90.000,E1 282.479} C_DIS
